# B&R Automation Studio project Soiled_PLC (part 11)

#### actGetServerReq.st
```iecst
(********************************************************************
 * COPYRIGHT --
 ********************************************************************
 * Program: hlKanLink
 * File: actGetServerReq.st
 * Author: stahlhut
 * Created: April 01, 2015
 ********************************************************************
 * Implementation of program hlKanLink
 ********************************************************************)

(* Kanlink Server/Request bearbeiten *)
ACTION actGetServerReq:
			// Commandos unter 1000 sind für alle gleich:
			IF Kanlink.ServerData.HeaderV1Rec.Command < 1000 THEN

				CASE Kanlink.ServerData.HeaderV1Rec.Command OF
					0:   // MaschinenInfo Senden: Darf jeder lesen

						Kanlink.ServerData.HeaderV1Send.Command := 1;
						Kanlink.ServerData.HeaderV1Send.dataFormat := 5;
						Kanlink.ServerData.HeaderV1Send.Length := 148;
						Kanlink.ServerData.HeaderV1Send.Tag := Kanlink.ServerData.HeaderV1Rec.Tag;
						Kanlink.ServerData.HeaderV1Send.ReqID := Kanlink.ServerData.HeaderV1Rec.ReqID;

						KLLib_SendData(ADR(Kanlink),ADR(Kanlink.ServerData.MetaInfoResp),SIZEOF(Kanlink.ServerData.MetaInfoResp),ADR(Kanlink.client_address));

					2:   // Response Ping: Darf jeder lesen

						Kanlink.ServerData.HeaderV1Send.Command := 3;
						Kanlink.ServerData.HeaderV1Send.dataFormat := 5;
						Kanlink.ServerData.HeaderV1Send.Length := 17;
						Kanlink.ServerData.HeaderV1Send.Tag := Kanlink.ServerData.HeaderV1Rec.Tag;
						Kanlink.ServerData.HeaderV1Send.ReqID := Kanlink.ServerData.HeaderV1Rec.ReqID;

						KLLib_SendData(ADR(Kanlink),ADR(Kanlink.ServerData.PingResp),SIZEOF(Kanlink.ServerData.PingResp),ADR(Kanlink.client_address));

				END_CASE;

			ELSE
					// >= 1000 sind spezifische Daten

					// Anfrage Konfiguriert?
					// Zur Anfrage Verbindung raussuchen..
					_xIdxFound := FALSE;
					_iIdxFound := 32000;

					KL_BuildKey(Command := Kanlink.ServerData.HeaderV1Rec.Command,CmdNr := UINT_TO_USINT( Kanlink.ServerData.HeaderV1Rec.CmdNr AND 16#000F) ,IPAdr := Kanlink.ServerData.IPAdr, adrKey:= ADR(Kanlink.RecKey));
					FOR _i := 0 TO HLKANLINK_MAX_SERVERCONNS  DO

						_ptrIndex ACCESS ADR(Kanlink.ServerListe[_i]);
						_dSrvIf ACCESS _ptrIndex.adrInterface;
						IF _ptrIndex.Adr = 0 THEN // wenn alle das Commando lesen dürfen/ Adresse und Area ausblenden
							IF Kanlink.RecKey.CmdKey = _ptrIndex.Key.CmdKey THEN // Index gefunden, beantworten:
								_xIdxFound := TRUE;
								_iIdxFound := _i;
								EXIT;
							END_IF;
						ELSE
							IF (Kanlink.RecKey.CmdKey = _ptrIndex.Key.CmdKey) AND (Kanlink.RecKey.IP_Key = _ptrIndex.Key.IP_Key) THEN // Index gefunden, beantworten:
								_xIdxFound := TRUE;
								_iIdxFound := _i;
								EXIT;
							END_IF;
						END_IF;
					END_FOR

					_xAdrErr := (_ptrIndex.AdrDataReq = 0) OR (_ptrIndex.AdrDataResp = 0);

					IF ( _xIdxFound = FALSE) OR _xAdrErr THEN // Falls keine gültige Verbindung dann Fehlerframe senden
						// Fehlerframe senden:
						Kanlink.ServerData.HeaderV1Send.Command := Kanlink.ServerData.HeaderV1Rec.Command +1;
						Kanlink.ServerData.HeaderV1Send.dataFormat := 255;
						Kanlink.ServerData.HeaderV1Send.Length := 68;
						Kanlink.ServerData.HeaderV1Send.Tag := Kanlink.ServerData.HeaderV1Rec.Tag;
						Kanlink.ServerData.HeaderV1Send.ReqID := Kanlink.ServerData.HeaderV1Rec.ReqID;

						// Error Frame:
						Kanlink.ServerData.ErrorFrame.ErrorNumber := 2;
						strcpy(ADR(Kanlink.ServerData.ErrorFrame.ErrorText),ADR('request not supported'));

						//	KLLib_SendData(ADR(Kanlink),ADR(Kanlink.ServerData.ErrorFrame),SIZEOF(Kanlink.ServerData.ErrorFrame),ADR(Kanlink.client_address));

					ELSE
						// Empfangene Daten speichern:

						IF NOT( (_dSrvIf.iState <> 0 )   AND _ptrIndex.xReqManually) THEN  // falls Req bereits bearbeitet wird verwerfen
							_ptrIndex.iReqCnt := _ptrIndex.iReqCnt + 1;
							_dSrvIf.iState := 1;
							strcpy(ADR(_ptrIndex.sClientIPAdr),ADR(Kanlink.client_address));
							// todo längenüberprüfung _ptrIndex.ReqLength
							memcpy(_ptrIndex.AdrDataReq,ADR(Kanlink.ServerData.receive_data)+PreHeaderSize+HeaderSize,_ptrIndex.ReqLength);

							_ptrIndex.iReqID := Kanlink.ServerData.HeaderV1Rec.ReqID;
							_dSrvIf.out.tag		:= Kanlink.ServerData.HeaderV1Rec.Tag;

							IF (_ptrIndex.CmdOpt AND KL_optOnReqCall) <> 0 THEN
								KL_OnRecReq(adrReqData := _ptrIndex.AdrDataReq, adrRespData := _ptrIndex.AdrDataResp, adrKanlink := ADR(Kanlink),_ptrIndex.Cmd, adrUserData := IFhlKanLink.Parameter.adrUserTyp );
							END_IF;
							IF _ptrIndex.xReqManually = 0 THEN

								Kanlink.ServerData.HeaderV1Send.Command := _ptrIndex.Cmd + 1;
								Kanlink.ServerData.HeaderV1Send.dataFormat := 5;
								Kanlink.ServerData.HeaderV1Send.Length := UDINT_TO_UINT( _ptrIndex.RespLength);
								Kanlink.ServerData.HeaderV1Send.ReqID := _ptrIndex.iReqID;
								Kanlink.ServerData.HeaderV1Send.CmdNr := _ptrIndex.CmdOpt AND 16#000F;
								Kanlink.ServerData.HeaderV1Send.Tag		:= _dSrvIf.tag;
								_ptrIndex.iConnectionTimer := 0;
								KLLib_SendData(ADR(Kanlink),_ptrIndex.AdrDataResp,_ptrIndex.RespLength,ADR(_ptrIndex.sClientIPAdr));
							END_IF;
						END_IF;

					END_IF;

			END_IF;

END_ACTION
```

#### actResponse.st
```iecst
(********************************************************************
 * COPYRIGHT --
 ********************************************************************
 * Program: hlKanLink
 * File: actResponse.st
 * Author: stahlhut
 * Created: April 01, 2015
 ********************************************************************
 * Implementation of program hlKanLink
 ********************************************************************)

(* Response eines Servers bearbeiten *)
ACTION actResponse:

			KL_BuildKey(Command := Kanlink.ServerData.HeaderV1Rec.Command,CmdNr := UINT_TO_USINT( Kanlink.ServerData.HeaderV1Rec.CmdNr AND 16#000F) ,IPAdr := Kanlink.ServerData.IPAdr, adrKey:= ADR(Kanlink.RecKey));

			_xIdxFound := FALSE;
			FOR _i := 0 TO HLKANLINK_MAX_CLIENTCONNS DO
				_dClient ACCESS ADR(Kanlink.ClientListe[_i]);

				IF (Kanlink.RecKey.CmdKey = _dClient.Key.CmdKey) AND (Kanlink.RecKey.IP_Key = _dClient.Key.IP_Key) THEN // Index gefunden, beantworten:
					_xIdxFound := TRUE;
					EXIT;
				END_IF;
			END_FOR

			_xAdrOK := _dClient.AdrDataResp <> 0 ;

			IF _xIdxFound AND _xAdrOK THEN
				_dClient.xReqPending := FALSE;
				IF _dClient.iTimeOutCnt > 0 THEN
					_dClient.iTimeOutCnt := _dClient.iTimeOutCnt - 1;
				END_IF;
				IF _dClient.adrInterface <> 0 THEN
					_dCltIf ACCESS _dClient.adrInterface;
					_dCltIf.iState := 3;
				END_IF;

				memcpy(_dClient.AdrDataResp,ADR(Kanlink.ServerData.receive_data) + PreHeaderSize+HeaderSize,_dClient.RespLength);
				_dCltIf.out.recTag := Kanlink.ServerData.HeaderV1Rec.Tag;

		  	END_IF;

			_iCltRespCnt := _iCltRespCnt + 1;
			Kanlink._xGetClientResp := FALSE;

			Kanlink._xSendClient := TRUE; // Daten einsortiert, nix weiter zutun also Clients bearbeiten
			Kanlink.udp.rec.enable := 1;

END_ACTION
```

### history.txt
```
1.00.3 horn 20.03.2017
hlKanLink wurde so erweitert, dass jetzt beim Server und Client eine beliebige IP-Adresse eingegeben werden kann.
AdvMode		Freischalten der Eingabe der gesamten IP-Adresse
AdrAdvMode	gesamte IP-Adresse der Gegenstelle.

1.00.2 horn 20.01.2016
Es werden jetzt keine Warnmeldungen mehr erzeugt.

1.00.1 sta 1.4.2015 sta
KG Framework - Kompatibel
Der Client kann nun einen UDINT Tag zum Server senden. Unterstützt der Server den Tag
wird ein Server-Tag zurückgesendet.
ifhlKanlink

0.94.5 sta 16.12.2014
udp_open mit IP-Adresse binden
27.3.12/sta/Struktur für Visualisierung

20.3.12/sta/Kommando Typen in einzelne Dateien geteilt
Compiler schalter "Autonom" eingefügt, Lib Autonom erstellt
Cmd WetExt angepasst

7.3.12/sta/version Kgframework
hlKanlink Version

21.02.12 sta 0.93
Client kann mit state gesteuert werden

8.2.12 sta 0.92
Fehler bei Server-Key behoben
2.2.12 sta
Zum einrichten eines Server und Client KLLib_CfgServer und KLLib_CfgClient integriert.
Konf sowohl über Parameter und mit den Funktionen möglich

30.1.12 sta
interface  umbenannt
MaxServerConn und MaxClientCon in userlib

todo:
"OneShot" Client-Statevariable
Überprüfung Längen der Commandos
Logger wieder inbetriebnehmen

Startversion 0.900
```

### Library Logical/KanLink_A19/KGFramework/Pkg_hlKanLink/KanLinkLib (IEC, version 0.94.5) - KanlinkHilfsfunktionen
Depends on: AsUDP, asstring, AsARCfg, brsystem, sys_lib, AsArLog, AsIODiag, AsETH, DataObj, KL_UserLib, KGstdLib

#### CmdBTxfer.typ - Commando Batch Transfer
```iecst
(********************************************************************
 * COPYRIGHT -- Herbert Kannegiesser GmbH
 ********************************************************************
 * Library: Kanlink Commando 1000 BatchTransfer
 * File:
 * Author: stahlhut
 * Created: 20.03.2012
 ********************************************************************
 * Data types of library WetLinkLib
 ********************************************************************)
(*Interne Strukturen*)

TYPE
	KL_BTxf_typ : 	STRUCT  (*Batch Transfer Server*)
		Req : KLreq1000_BTH_typ;
		Resp : KLresp1000_BTH_typ;
	END_STRUCT;
	KLreq1000_BTH_typ : 	STRUCT
		xHready : BOOL;
		xHreadyForLoad : BOOL;
		xHbatchReceived : BOOL;
		xHtransferzoneOccupied : BOOL;
		xHreqCtrlTransfer : BOOL;
		xHtransferRunning : BOOL;
		xHwaitingForTransfer : BOOL;
		xHshiftBatches : BOOL;
		wHstate : UINT;
		xHcmdAutomatic : BOOL;
		xHreserve : ARRAY[1..5]OF BOOL;
		wTimeToReadyForLoad : UINT;
		wRemainProctime : UINT; (*Remaining Processtime / Verbleibende Prozesszeit*)
	END_STRUCT;
	KLresp1000_BTH_typ : 	STRUCT
		xHsCmdFinishProcess : BOOL;
		xHsReqForUnload : BOOL;
		xHsUnloading : BOOL;
		xHsReqCtrlTransfer : BOOL;
		xHsTransferRunning : BOOL;
		xHsRes : BOOL;
		wState : UINT;
		xCmdAuto : BOOL;
		xCmdStartProcess : BOOL;
		xHsDataValid : BOOL;
		xHsRes2 : ARRAY[0..2]OF BOOL;
		wCntLoads : UINT;
		BatchData : BatchData_typ;
	END_STRUCT;
END_TYPE
```

#### KLInterface.typ - Interfacetypen Kanlink
```iecst
(********************************************************************
 * COPYRIGHT -- Herbert Kannegiesser GmbH
 ********************************************************************
 * Library: Kanlink	 Interface
 * File:
 * Author: stahlhut
 * Created: 20.03.2012
 ********************************************************************
 * Data types of Interface Kanlink
 ********************************************************************)

TYPE
	KL_Key_typ : 	STRUCT
		IP_Key : UDINT;
		CmdKey : UDINT;
	END_STRUCT;
	KL_Parameter_typ : 	STRUCT
		Server : ARRAY[0..HLKANLINK_MAX_SERVERCONNS]OF KL_ServerPar_typ;
		Client : ARRAY[0..HLKANLINK_MAX_CLIENTCONNS]OF KL_ClientPar_typ;
		adrUserTyp : UDINT;
	END_STRUCT;
	KL_ClientPar_typ : 	STRUCT
		Name : STRING[15];
		Adr : UINT;
		Cmd : UINT;
		CmdOpt : UINT; (*Bits 0..3 = Nummer des Clients*)
		Area : UINT;
		CycleTime : UINT;
		sReq : STRING[80];
		sResp : STRING[80];
		AdvMode : BOOL; (*Modus mit dem eine vollständige IP-Adresse eingegeben werden kann*)
		AdrAdvMode : STRING[16]; (*Vollständige IP-Adresse*)
	END_STRUCT;
	KL_ServerPar_typ : 	STRUCT
		Name : STRING[15];
		Adr : UINT;
		Cmd : UINT;
		CmdOpt : UINT; (*Bits 0..3 = Nummer der Verbindung*)
		Area : UINT;
		TimeOut : UINT;
		sReq : STRING[80];
		sResp : STRING[80];
		AdvMode : BOOL; (*Modus mit dem eine vollständige IP-Adresse eingegeben werden kann
oder die Prüfung der IP-Adresse entfällt.*)
		AdrAdvMode : STRING[16]; (*Vollständige IP-Adresse*)
	END_STRUCT;
	IF_ServerOutTyp : 	STRUCT
		xConnected : BOOL;
		iCfgState : UINT; (*0 = ConfOK*)
		tag : UDINT;
	END_STRUCT;
	IF_Server_typ : 	STRUCT
		iState : UINT;
		out : IF_ServerOutTyp;
		tag : UDINT;
	END_STRUCT;
	IF_ClientOut_typ : 	STRUCT
		xConnected : BOOL;
		recTag : UDINT;
	END_STRUCT;
	IF_Client_typ : 	STRUCT
		out : IF_ClientOut_typ;
		iState : UINT;
		tag : UDINT;
	END_STRUCT;
	IFhlKanLink_Typ : 	STRUCT
		in : IF_KL_Control_in_typ;
		Server : ARRAY[0..HLKANLINK_MAX_SERVERCONNS]OF IF_Server_typ;
		Client : ARRAY[0..HLKANLINK_MAX_CLIENTCONNS]OF IF_Client_typ;
		Parameter : KL_Parameter_typ;
		xError : BOOL; (*Kanlink in Störung*)
	END_STRUCT;
	IF_KL_Control_in_typ : 	STRUCT
		xRun : BOOL; (*Rise= Starten Kanlink /fall = stoppen Kanlink*)
		xRestart : BOOL;
	END_STRUCT;
	IF_KL_Control_out_typ : 	STRUCT
		iError : UINT;
		iServerError : ARRAY[0..HLKANLINK_MAX_SERVERCONNS]OF UINT;
		iClientError : ARRAY[0..HLKANLINK_MAX_CLIENTCONNS]OF UINT;
		iStep : UINT; (*Statemachine KanLink*)
	END_STRUCT;
	IFhlKLVisuIN_typ : 	STRUCT
		cmdNr : INT; (*Ausführbares Commando*)
		cmdTag : INT; (*Dazugehörige Daten*)
		iServerNr : UINT; (*zu lesende Serverlist*)
		iCltNr : UINT; (*zu lesender Client*)
	END_STRUCT;
	IFhlKLVisuOUT_typ : 	STRUCT
		step : UINT;
		udpOpenStatus : UINT;
		udpSendStatus : UINT;
		udpRecStatus : UINT;
		iCycleTime : UINT;
		udNetId : UDINT;
		server : KL_ServerListe_typ;
		client : KL_ClientListe_typ;
		cmdResp : INT; (*Response auf CmdNr*)
	END_STRUCT;
	IFhlKLVisu_typ : 	STRUCT
		in : IFhlKLVisuIN_typ;
		out : IFhlKLVisuOUT_typ;
	END_STRUCT;
END_TYPE
```

#### KanLinkLib.typ - Exported data types
```iecst
(********************************************************************
 * COPYRIGHT -- Herbert Kannegiesser GmbH
 ********************************************************************
 * Library: WetLinkLib
 * File: WetLinkLib.typ
 * Author: stahlhut
 * Created: January 06, 2012
 ********************************************************************
 * Data types of library WetLinkLib
 ********************************************************************)
(*Interne Strukturen*)

TYPE
	udp_typ : 	STRUCT  (*UDP Typ*)
		open : UdpOpen;
		send : UdpSend;
		rec : UdpRecv;
		close : UdpClose;
	END_STRUCT;
	udint_array_typ : 	STRUCT  (*Casten von UDINT -> byte*)
		a : USINT;
		b : USINT;
		c : USINT;
		d : USINT;
	END_STRUCT;
	ServerDataTyp : 	STRUCT  (*Datatyp for global Variables*)
		receive_data : ARRAY[0..8191]OF USINT; (*Data which has been received*)
		send_data : ARRAY[0..8191]OF USINT; (*Data which should be sent*)
		PreHeaderSend : PreHeader_Typ;
		PreHeaderRec : PreHeader_Typ;
		HeaderV1Send : HeaderV1_Typ;
		HeaderV1Rec : HeaderV1_Typ;
		MetaInfoResp : KLresp0_MetaInfo_typ;
		ErrorFrame : KL_Error_Frame_typ;
		PingReq : KLreq2_Ping_typ;
		PingResp : KLresp2_Ping_typ;
		IPAdr : STRING[16]; (*IP-Adresse des Clients*)
	END_STRUCT;
	PreHeader_Typ : 	STRUCT
		Magic : UDINT; (*MagicNr*)
		HeaderVersion : UINT; (*Headerversion*)
		Tag : UINT; (*Reserve*)
	END_STRUCT;
	HeaderV1_Typ : 	STRUCT
		ReqID : UINT;
		dataFormat : UINT;
		Command : UINT;
		Length : UINT;
		CmdNr : UINT;
		CmdTag : UINT; (*Unterschiedliche Parameter zum Command*)
		Tag : UDINT; (*Reserve/Spezial*)
	END_STRUCT;
	KL_ServerListe_typ : 	STRUCT
		Cmd : UINT;
		CmdOpt : UINT;
		Adr : UINT;
		Area : UINT;
		pRespStr : UDINT; (*Adresse des Resp String*)
		pReqStr : UDINT; (*Adresse des Req String*)
		AdrDataReq : UDINT;
		ReqLength : UDINT; (*Länge Request Daten*)
		AdrDataResp : UDINT;
		RespLength : UDINT; (*Länge Response Daten*)
		Key : KL_Key_typ; (*Suchschlüssel/ Darf nicht doppelt vorkommen== Konfigurierungsfehler*)
		xConnected : BOOL; (*Falls Commando 2s nicht angefragt wird ist verbindung unterbrochen*)
		iConnectionTimer : UINT; (*Der Zugehörige Zähler / Timer*)
		adrParameter : UDINT; (*Adresse der Parameter*)
		sServerIPAdr : STRING[16];
		sClientIPAdr : STRING[16];
		iReqCnt : UINT;
		xReqManually : BOOL;
		iReqID : UINT;
		iCfgStatus : UINT;
		adrInterface : UDINT;
		xActiv : BOOL;
		tag : UDINT;
	END_STRUCT;
	KL_ClientListe_typ : 	STRUCT
		RecCmd : UINT; (*Rec Command nr*)
		Cmd : UINT; (*Send Command nr*)
		CmdOpt : UINT; (*SendeOptionen Senden Nr des Commando etc*)
		Adr : UINT;
		Area : UINT;
		Key : KL_Key_typ;
		pResp : UDINT; (*Adresse des Namen der Response Struktur*)
		pReq : UDINT; (*Adresse des Namen der Request Struktur*)
		AdrDataReq : UDINT;
		AdrDataResp : UDINT;
		ReqLength : UDINT;
		RespLength : UDINT;
		TimeOut : UINT;
		TimeOutLeft : UINT;
		xError : BOOL;
		iCycleWait : UINT;
		iCycleTime : UINT;
		xDataRec : BOOL;
		iReqId : UINT;
		sClientAdr : STRING[16];
		xReqPending : BOOL;
		iTimeOutCnt : UINT;
		xActiv : BOOL;
		iCnt : UINT;
		xConnected : BOOL; (*True wenn Verbindung aktiv und läuft*)
		iTimeOutCnt_Summe : UINT;
		adrInterface : UDINT;
		adrParameter : UDINT; (*Adresse der Parameter*)
		recTag : UDINT; (*Tag des Kommandos*)
	END_STRUCT;
END_TYPE

(*Kommandos*)

TYPE
	BatchData_typ : 	STRUCT
		dtTimeStamp : DATE_AND_TIME;
		bTypeBatchNo : USINT;
		bCntCustomers : USINT;
		wTotalWeight : UINT;
		bBatchNo : ARRAY[0..15]OF USINT;
		sCategory : STRING[11];
		utfMark : ARRAY[0..31]OF UINT;
		bCustom : ARRAY[0..11]OF USINT;
		PartBatch : ARRAY[0..7]OF PartBatchData_typ;
	END_STRUCT;
	PartBatchData_typ : 	STRUCT
		sCustomNo : STRING[11];
		wCustomWeight : UINT;
	END_STRUCT;
	KL_Error_Frame_typ : 	STRUCT
		Version : UINT;
		ErrorNumber : UINT;
		ErrorText : STRING[63];
	END_STRUCT;
	KLresp0_MetaInfo_typ : 	STRUCT
		KanLink_Hostname : STRING[15];
		Machine_type : STRING[15];
		SoftwareNo : STRING[15];
		SoftwareVersion : STRING[15];
		DataModelTimeStamp : DATE_AND_TIME;
		DataModelVersion : UINT;
		TimeZone : UINT;
		SommerTime : UINT;
	END_STRUCT;
	KLreq2_Ping_typ : 	STRUCT
		KanLink_Hostname : STRING[15];
	END_STRUCT;
	KLresp2_Ping_typ : 	STRUCT
		KanLink_Hostname : STRING[15];
		FrameVersion : USINT;
	END_STRUCT;
END_TYPE
```

#### KanLinkLib.fun - Exported functions and function blocks
```iecst
(********************************************************************
 * COPYRIGHT -- Herbert Kannegiesser GmbH
 ********************************************************************
 * Library: WetLinkLib
 * File: WetLinkLib.fun
 * Author: stahlhut
 * Created: January 06, 2012
 ********************************************************************
 * Functions and function blocks of library WetLinkLib
 ********************************************************************)

FUNCTION_BLOCK KanLink_FB (*TODO: Add your comment here*)
	VAR_INPUT
		Step : UINT; (*state machine*)
		ErrorNr : UINT;
		client_address : STRING[16]; (*Speichern der Receiver Adresse*)
		RecKey : KL_Key_typ;
		sNetID : STRING[15];
		udNetID : UDINT;
		udp : udp_typ;
		ServerData : ServerDataTyp;
		ServerListe : ARRAY[0..HLKANLINK_MAX_SERVERCONNS] OF KL_ServerListe_typ; (*Erlaubte Daten Server*)
		ClientListe : ARRAY[0..HLKANLINK_MAX_CLIENTCONNS] OF KL_ClientListe_typ;
		_xOpenPort : BOOL;
		_xSendClient : BOOL;
		_xGetClientResp : BOOL;
		_xGetServerReq : BOOL;
		_uiLastId : UDINT;
		CanReturn : BOOL;
		adrSelf : UDINT; (*Eigene Adresse, zum weiterleiten an Function/Function Block*)
		_offset : UDINT; (*Offset zum Berechnen der Sendelänge*)
		_SendLen : UDINT; (*Sendelänge*)
		DoCommand : UINT;
		KLLib_Init_0 : KLLib_Init;
		_iCycleTime : UINT;
		adrInterface : UDINT;
		iPort : UINT; (*Port nr (23500)*)
		sIF : STRING[10]; (*Interface Ethernet*)
		CfgClient : KLLib_CfgClient;
		CfgServer : KLLib_CfgServer;
	END_VAR
	VAR_OUTPUT
		xReturn : BOOL;
	END_VAR
	VAR
		_dPrehead : REFERENCE TO PreHeader_Typ;
		_dHead : REFERENCE TO HeaderV1_Typ;
		_udArr : REFERENCE TO udint_array_typ;
		_dRecAdr : UDINT;
		_xPreheadOK : BOOL;
		_xVersionOK : BOOL;
		_xUse : BOOL;
	END_VAR
END_FUNCTION_BLOCK

FUNCTION KLLib_ClientTimer : BOOL (*Bearbeitet Timeout und Cycletime (Zähler)*)
	VAR_INPUT
		Srv : REFERENCE TO KanLink_FB;
		_iCycleTime : UINT;
	END_VAR
	VAR
		_dClient : REFERENCE TO KL_ClientListe_typ;
		_i : UINT;
		_dServer : REFERENCE TO KL_ServerListe_typ;
		_dInterface : REFERENCE TO IF_Client_typ;
		_dSrvIf : REFERENCE TO IF_Server_typ;
	END_VAR
END_FUNCTION

FUNCTION KLLib_GetPVAdr : UDINT (*Adresse der PV ermitteln (Server)*)
	VAR_INPUT
		ServerItem : REFERENCE TO KL_ServerListe_typ;
	END_VAR
	VAR
		iStat : INT;
	END_VAR
END_FUNCTION

FUNCTION KLLib_SendData : UDINT (*TODO: Add your comment here*)
	VAR_INPUT
		Srv : REFERENCE TO KanLink_FB;
		SendAdr : UDINT;
		SendLen : UDINT;
		pDestination : UDINT; (*Adresse des Zielstrings*)
	END_VAR
END_FUNCTION

FUNCTION KLLib_ReadServerPara : UDINT (*TODO: Add your comment here*)
	VAR_INPUT
		adrServerItem : UDINT;
		adrParaItem : UDINT;
		adrKanLink : UDINT;
	END_VAR
	VAR
		_xError : BOOL;
		KanLink : REFERENCE TO KanLink_FB;
		dServer : REFERENCE TO KL_ServerListe_typ;
		dPara : REFERENCE TO KL_ServerPar_typ;
		_udAdr : UDINT;
		_udArr : REFERENCE TO udint_array_typ;
		_udNetId : REFERENCE TO udint_array_typ;
	END_VAR
END_FUNCTION

FUNCTION KLLib_ReadClientPara : UDINT (*TODO: Add your comment here*)
	VAR_INPUT
		adrClientItem : UDINT;
		adrParaItem : UDINT;
		adrServer : UDINT;
	END_VAR
	VAR
		_xError : BOOL;
		dClient : REFERENCE TO KL_ClientListe_typ;
		dPara : REFERENCE TO KL_ClientPar_typ;
		_udArr : REFERENCE TO udint_array_typ;
		_udAdr : UDINT;
		dServer : REFERENCE TO KanLink_FB;
		_udNetId : REFERENCE TO udint_array_typ;
	END_VAR
END_FUNCTION

FUNCTION KLLib_InitCltPV : UDINT (*TODO: Add your comment here*)
	VAR_INPUT
		dclt : REFERENCE TO KL_ClientListe_typ;
	END_VAR
	VAR
		iStat : UINT;
	END_VAR
END_FUNCTION

FUNCTION_BLOCK KLLib_Init (*TODO: Add your comment here*)
	VAR_INPUT
		enable : BOOL;
		adrServer : UDINT;
		adrInterface : UDINT;
	END_VAR
	VAR_OUTPUT
		status : UINT;
	END_VAR
	VAR
		_bStep : INT;
		_dServer : REFERENCE TO KanLink_FB;
		GetEthPort_0 : kgGetEthPort;
		CfgGetIPAddr_0 : CfgGetIPAddr;
		RTInfo_0 : RTInfo;
		_i : INT;
		_dIf : REFERENCE TO IFhlKanLink_Typ;
	END_VAR
END_FUNCTION_BLOCK

FUNCTION KL_BuildKey : BOOL
	VAR_INPUT
		Command : UINT;
		CmdNr : USINT;
		IPAdr : STRING[16];
		adrKey : UDINT;
	END_VAR
	VAR
		IP_Key : UDINT;
		Key : REFERENCE TO KL_Key_typ;
	END_VAR
END_FUNCTION

FUNCTION_BLOCK KLLib_CfgClient (*Configuriert einen Kanlink Client*)
	VAR_INPUT
		adrKanlink : UDINT;
		ClientIndex : UINT;
		adrName : UDINT;
		IPAdr : USINT;
		Area : USINT;
		CmdOpt : UINT;
		Cmd : UINT;
		CycleTime : UINT;
		adrSReq : UDINT;
		adrSResp : UDINT;
	END_VAR
	VAR_OUTPUT
		status : UINT;
	END_VAR
	VAR
		_dKL : REFERENCE TO KanLink_FB;
		_dCltPar : REFERENCE TO KL_ClientPar_typ;
		_iret : UDINT;
	END_VAR
END_FUNCTION_BLOCK

FUNCTION_BLOCK KLLib_CfgServer (*Configuriert einen Kanlink Server*)
	VAR_INPUT
		adrKanlink : UDINT;
		ServerIndex : UINT;
		adrName : UDINT;
		IPAdr : USINT;
		Area : USINT;
		CmdOpt : UINT;
		Cmd : UINT;
		TimeOut : UINT;
		adrSReq : UDINT;
		adrSResp : UDINT;
	END_VAR
	VAR_OUTPUT
		status : UINT;
	END_VAR
	VAR
		_dKL : REFERENCE TO KanLink_FB;
		_dSrvPar : REFERENCE TO KL_ServerPar_typ;
		_iret : UDINT;
	END_VAR
END_FUNCTION_BLOCK

FUNCTION KLLib_CreateStrucDef : UINT (*Erzeuge eine Strukturdefinition zu einer Variablen*)
	VAR_INPUT
		lPtrAdr : UDINT;
		lPtrLen : UDINT;
		sRootName : STRING[127];
		sItemName : STRING[31];
		lDataAdr : UDINT;
	END_VAR
	VAR
		_wStatus : UINT;
		_sPvName : STRING[127];
		_lDataType : UDINT;
		_lDataLen : UDINT;
		_wDataDimension : UINT;
		_sLine : STRING[127];
		_sValueLen : STRING[11];
		_lAdr : REFERENCE TO UDINT;
		_lLen : REFERENCE TO UDINT;
		_sValueDim : STRING[5];
		_sValueOffs : STRING[11];
		_i : UINT;
		_sItemName : STRING[31];
		_sType : ARRAY[1..23] OF STRING[15] := ['BOOL','SINT','INT','DINT','USINT','UINT','UDINT','REAL','STRING','ULINT','DATE_AND_TIME','TIME','DATE','LREAL','','TIME_OF_DAY','BYTE','WORD','DWORD','LWORD','WSTRING','','LINT'];
		_lDataAdr : UDINT;
	END_VAR
END_FUNCTION

FUNCTION KLLib_WriteStrucDefLine : UINT (*Übertrage einen String als Zeile in den Speicher*)
	VAR_INPUT
		lPtrLine : UDINT;
		lPtrAdr : UDINT;
		lPtrLen : UDINT;
	END_VAR
	VAR
		_lAdr : REFERENCE TO UDINT;
		_lLen : REFERENCE TO UDINT;
		_iStringlen : INT;
		_sLine : REFERENCE TO STRING[127];
	END_VAR
END_FUNCTION
```

#### KanLink_FB.st - core-Funktion
```iecst
(********************************************************************
 * COPYRIGHT -- Herbert Kannegiesser GmbH
 ********************************************************************
 * Library: Kanlink
 * File:
 * Author: stahlhut
 * Created: January 06, 2012
 ********************************************************************
 * Implementation of library Kanlink

29.8.2012 Bug behoben verunden recAdr mit 0x0F

 ********************************************************************)

FUNCTION_BLOCK KanLink_FB

	xReturn := 0;

	IF Step <> 10 THEN
		xReturn := 1;
		RETURN;
	END_IF;
	KLLib_ClientTimer(adrSelf,_iCycleTime);

	IF  udp.send.enable THEN
		udp.send;

		IF  udp.send.status = 0 THEN
			udp.send.enable := FALSE;
		ELSIF udp.send.status = ERR_FUB_BUSY THEN
			udp.send.enable := TRUE;
			xReturn := 1;
			RETURN;
		ELSE
			ErrorNr := 4;
			udp.send.enable := FALSE;
		END_IF
	END_IF;

	udp.rec.enable := 1;
	udp.rec.ident := udp.open.ident;
	udp.rec.pData := ADR(ServerData.receive_data);	// Datenspeicher
	udp.rec.datamax := SIZEOF(ServerData.receive_data);	// Länge des Datenspeichers
	udp.rec.flags := 0;
	udp.rec.pIpAddr := ADR(client_address);	// IP Adresse des Senders
	udp.rec;

	IF udp.rec.status = 0 THEN  // Daten empfangen
		// Header Daten kopieren
		_dPrehead ACCESS ADR(ServerData.receive_data);
		_dHead ACCESS ADR(ServerData.receive_data) + PreHeaderSize;
		memcpy(ADR(ServerData.PreHeaderRec),ADR(ServerData.receive_data),PreHeaderSize);
		memcpy(ADR(ServerData.HeaderV1Rec),ADR(ServerData.receive_data)+PreHeaderSize,SIZEOF(ServerData.HeaderV1Rec));

		ServerData.IPAdr := client_address;

		_xPreheadOK := (ServerData.PreHeaderRec.Magic = MagicNr);
		_xVersionOK := (ServerData.PreHeaderRec.HeaderVersion = 16#100);

		IF (_dHead.Command AND 1) = 0 THEN
			_xGetServerReq := TRUE;
		ELSIF (_dHead.Command AND 1) = 1 THEN
			_xGetClientResp := TRUE;
		END_IF;

	ELSIF udp.rec.status = udpERR_NO_DATA THEN  // Keine Daten empfangen, Client abarbeiten
		_xSendClient := TRUE;
	ELSIF udp.rec.status = ERR_FUB_BUSY THEN  (* UdpRecv not finished -> redo *)
		xReturn := 1;
		RETURN;
	ELSE  (* Goto Error Step *)
		ErrorNr := 5;
		xReturn := 1;
		RETURN;
	END_IF

	// dieser teil ist nur für den Linker (unused Variable)
	IF _xUse THEN
		RecKey := RecKey;
		sNetID := sNetID;
		udNetID := udNetID;
		ServerListe := ServerListe;
		ClientListe	:= ClientListe;
		_xOpenPort := _xOpenPort;
		_uiLastId	:= _uiLastId;
		CanReturn	:= CanReturn;
		_offset 	:= _offset;
		_SendLen	:= _SendLen;
		DoCommand	:= DoCommand;
	 	adrInterface	:= adrInterface;
		iPort 	:= iPort;
		sIF	:= sIF;
		KLLib_Init_0.enable	:= KLLib_Init_0.enable;
		CfgClient.adrKanlink	:= CfgClient.adrKanlink;
		CfgServer.adrKanlink	:= CfgServer.adrKanlink;
	END_IF;

END_FUNCTION_BLOCK
```

#### KLLib_ClientTimer.st
```iecst
(********************************************************************
 * COPYRIGHT -- Herbert Kannegiesser GmbH
 ********************************************************************
 * Library: WetLinkLib
 * File: WLLIb_ClientTimer.st
 * Author: stahlhut
 * Created: January 06, 2012
 ********************************************************************
 * Implementation of library WetLinkLib
 ********************************************************************)

(* TODO: Add your comment here *)
FUNCTION KLLib_ClientTimer
FOR _i := 0 TO HLKANLINK_MAX_CLIENTCONNS DO
	_dClient  ACCESS ADR(Srv.ClientListe[_i]);
	_dInterface ACCESS (_dClient.adrInterface);

	// TimeOut (kurz) taskgerecht berechnen
	IF (_dClient.TimeOutLeft >= _iCycleTime) AND _dClient.xReqPending THEN
 		_dClient.TimeOutLeft := _dClient.TimeOutLeft - _iCycleTime;
	END_IF;

	IF _dClient.iCycleWait <= _dClient.iCycleTime THEN
		_dClient.iCycleWait := _dClient.iCycleWait + _iCycleTime;
	END_IF;
	// Timeout aufgetreten nur bis n Zählen. Retry sofort nach timeout, sonst retry nach cycletime
	IF _dClient.xReqPending AND (_dClient.TimeOutLeft < _iCycleTime) THEN
		_dClient.iTimeOutCnt_Summe := _dClient.iTimeOutCnt_Summe + 1;
		_dClient.xReqPending := FALSE;	// noch mal versuchen
		IF _dClient.iTimeOutCnt < 5 THEN
			_dClient.iTimeOutCnt := _dClient.iTimeOutCnt +1 ;
			_dClient.xReqPending := FALSE;	// noch mal versuchen
			_dInterface.iState := 4;
			_dClient.iCycleWait := _dClient.iCycleTime;
		END_IF;
	END_IF;
		// Verbindungsfehler
	_dClient.xConnected := (_dClient.iTimeOutCnt < 5) AND _dClient.xActiv AND (_dClient.iCycleTime > 0);
	_dInterface.out.xConnected := _dClient.xConnected;
	IF (_dClient.iTimeOutCnt >= 5 ) AND ( _dInterface.iState = 2 ) THEN
		_dInterface.iState := 255; // Timeout melden
	END_IF;

END_FOR;

FOR _i := 0 TO HLKANLINK_MAX_SERVERCONNS DO
	_dServer ACCESS ADR(Srv.ServerListe[_i]);
	_dSrvIf ACCESS _dServer.adrInterface;

	IF _dServer.iConnectionTimer <= 2000 THEN
		_dServer.iConnectionTimer := _dServer.iConnectionTimer + _iCycleTime;
	END_IF;
	_dServer.xConnected := (_dServer.iConnectionTimer < 2000);
	_dSrvIf.out.xConnected := _dServer.xConnected;
END_FOR;
KLLib_ClientTimer := 0;

END_FUNCTION
```

#### KLLib_SendData.st
```iecst
(********************************************************************
 * COPYRIGHT -- Herbert Kannegiesser GmbH
 ********************************************************************
 * Library: WetLinkLib
 * File: WLLib_SendData.st
 * Author: stahlhut
 * Created: January 07, 2012
 * changed April 2015
 ********************************************************************
 *
 ********************************************************************)

FUNCTION KLLib_SendData
	IF Srv.udp.send.enable = TRUE THEN //Sendung noch unterwegs, abbrechen
 		KLLib_SendData := 1;
		RETURN;
	END_IF;

	Srv.ServerData.PreHeaderSend.Magic := MagicNr;
	Srv.ServerData.PreHeaderSend.HeaderVersion := 16#0100;
	Srv._offset := 0;
	memcpy(ADR(Srv.ServerData.send_data),ADR(Srv.ServerData.PreHeaderSend),PreHeaderSize);
	Srv._offset := PreHeaderSize;

	memcpy(ADR(Srv.ServerData.send_data)+Srv._offset,ADR(Srv.ServerData.HeaderV1Send),HeaderSize);
	Srv._offset := Srv._offset+ HeaderSize;
	memcpy(ADR(Srv.ServerData.send_data)+Srv._offset,SendAdr,SendLen);
	Srv._SendLen := Srv._offset + Srv.ServerData.HeaderV1Send.Length;

	// Telegramm jetzt senden
	Srv.udp.send.enable := 1;
	Srv.udp.send.ident 	:= Srv.udp.open.ident;	(* Client Ident from AsUDP.UDP_Open *)
	Srv.udp.send.pHost 	:= pDestination;	(* IP Address of the Client *)
	Srv.udp.send.port 	:= Srv.iPort;
	Srv.udp.send.pData 	:= ADR(Srv.ServerData.send_data);	(* Which data to send *)
	Srv.udp.send.datalen :=  Srv._SendLen; //
	Srv.udp.send.flags 	:= 0;
	Srv.udp.send ;	(* Call the Function*)

END_FUNCTION
```

#### KL_BuildKey.st - Berechnen des Connection Key
```iecst
(********************************************************************
 * COPYRIGHT -- Herbert Kannegiesser GmbH
 ********************************************************************
 * Library: KanLinkLib
 * Datei: KL_BuildKey.st
 * Autor: stahlhut
 * Erstellt: 16. Januar 2012
 ********************************************************************
 * Implementierung der Library KanLinkLib
 ********************************************************************)

(* Berechnen des Connection Key *)
FUNCTION KL_BuildKey

	IF adrKey = 0 THEN // Fehler aufgetreten

		Key.CmdKey := 0;
		Key.IP_Key := 0;
		KL_BuildKey := FALSE;

	ELSE

		Key ACCESS adrKey;
		Key.CmdKey := SHL(UINT_TO_UDINT(Command),4)+USINT_TO_UINT(CmdNr);
		ethInetAton(ADR(IPAdr),ADR(IP_Key));
		Key.IP_Key := IP_Key;
		KL_BuildKey := TRUE;

	END_IF

END_FUNCTION
```

#### KLLib_Init.st
```iecst
(********************************************************************
 * COPYRIGHT -- Herbert Kannegiesser GmbH
 ********************************************************************
 * Library: KanLinkLib
 * File: KL_Init.st
 * Author: stahlhut
 * Created: January 12, 2012
 ********************************************************************
 * Implementation of library KanLinkLib
 ********************************************************************)

(* TODO: Add your comment here *)
FUNCTION_BLOCK KLLib_Init

	IF (adrServer = 0) OR (adrInterface = 0 )  THEN // fehler
		status := 1;
		enable := 0;
		RETURN;
	END_IF;
	IF enable = 0 THEN
		status := ERR_FUB_ENABLE_FALSE;
		RETURN;
	END_IF;

	IF (status = ERR_FUB_BUSY	) AND (enable = 0) THEN
		status := ERR_FUB_ENABLE_FALSE;
		_bStep := 100;
	END_IF;

	CASE _bStep OF
		0: // nix tun
			status := ERR_FUB_BUSY;
			_bStep := 10;
		10:
			_dServer ACCESS adrServer;
			_dServer.adrSelf := adrServer;
			_dIf ACCESS adrInterface;
			_dServer.adrInterface := adrInterface;

			IF _dServer.iPort = 0 THEN
				_dServer.iPort := 23500; // standardport benutzen
			END_IF;
			RTInfo_0.enable := TRUE;
			RTInfo_0;

			_dServer._iCycleTime := UDINT_TO_UINT( RTInfo_0.cycle_time / 1000);

			_bStep := 20;
		20:
			GetEthPort_0.enable := 1;
			GetEthPort_0.adrIF := ADR(_dServer.sIF);
			GetEthPort_0;
			IF GetEthPort_0.status = ERR_OK THEN
				_bStep := 30;
			ELSIF GetEthPort_0.status <> ERR_FUB_BUSY THEN // fehler aufgetreten
				status := 2;
				_bStep := 100;
			END_IF;
		30:
			CfgGetIPAddr_0.enable  := 1;
			CfgGetIPAddr_0.pDevice := ADR(_dServer.sIF);
			CfgGetIPAddr_0.pIPAddr := ADR(_dServer.sNetID);
			CfgGetIPAddr_0.Len := 16;
			CfgGetIPAddr_0;
			IF  (CfgGetIPAddr_0.status = ERR_OK) THEN
				_bStep := 40;
				ethInetAton(ADR(_dServer.sNetID),ADR(_dServer.udNetID));

			ELSIF CfgGetIPAddr_0.status <> ERR_FUB_BUSY THEN // fehler aufgetreten
				status := 3;
				_bStep := 100;
			END_IF;

		40:
			FOR _i := 0 TO HLKANLINK_MAX_SERVERCONNS DO
				_dServer.ServerListe[_i].adrInterface := ADR(_dIf.Server[_i]);
				KLLib_ReadServerPara(ADR(_dServer.ServerListe[_i]), ADR( _dIf.Parameter.Server[_i]),ADR(_dServer));
			END_FOR;
			//			memset(ADR(_dServer.ClientListe),0,SIZEOF(_dServer.ClientListe));
			FOR _i := 0 TO HLKANLINK_MAX_CLIENTCONNS DO
				KLLib_ReadClientPara(ADR(_dServer.ClientListe[_i]),ADR(_dIf.Parameter.Client[_i]),ADR(_dServer));
				_dServer.ClientListe[_i].xActiv := (_dServer.ClientListe[_i].Cmd <> 0);
				_dServer.ClientListe[_i].TimeOut := 140;
				_dServer.ClientListe[_i].adrInterface := ADR(_dIf.Client[_i]);
			END_FOR;
			_bStep := 50;
		50:

			_dServer.udp.open.enable := 1;
			_dServer.udp.open.pIfAddr := ADR(_dServer.sNetID);	(* Übergeben des Interface funzt nicht *)
			_dServer.udp.open.port := _dServer.iPort;	(* Port to listen*)
			_dServer.udp.open.options := 0;
			_dServer.udp.open;	(* Call the Function*)

			IF _dServer.udp.open.status = 0 THEN  (* UdpOpen successful*)
				_dServer._uiLastId := _dServer.udp.open.ident;
				_bStep := 90;
			ELSIF _dServer.udp.open.status = ERR_FUB_BUSY THEN  (* UdpOpen not finished -> redo *)

			ELSIF _dServer.udp.open.status = udpERR_ALREADY_EXIST THEN // erst schliessen
				_dServer.udp.close.enable := 1;
				_dServer.udp.close.ident := _dServer._uiLastId;
				_dServer.udp.close;
				IF _dServer.udp.close.status = 0 THEN
					//
				ELSIF _dServer.udp.close.status = ERR_FUB_BUSY THEN

				ELSE
					status := 5001;
					_bStep := 100;	// unbekannter close fehler aufgetreten
				END_IF;

			ELSE
				status := 5002;
				_bStep := 100; // unbekannter open fehler aufgetreten
			END_IF

		90:  // fertig
			status := ERR_OK;
			enable := 0;
			_bStep := 0;

		100: // fehler aufgetreten
			enable := 0;
			_bStep := 0;

	END_CASE;

END_FUNCTION_BLOCK
```

### Package Logical/KanLink_A19/KGFrameworkShare - Benutzereinstellungen


### Package Logical/KanLink_A19/KGFrameworkShare/Pkg_hlKanLinkUser - Kanlink User

### Library Logical/KanLink_A19/KGFrameworkShare/Pkg_hlKanLinkUser/KL_UserLib (IEC, version 0.91.0) - Kanlink User Library

#### KL_UserLib.var - Exported constants
```iecst
(********************************************************************
 * COPYRIGHT -- Herbert Kannegiesser GmbH
 ********************************************************************
 * Library: WL_UserLib
 * File: WL_UserLib.var
 * Author: stahlhut
 * Created: January 10, 2012
 ********************************************************************
 * Constants of library WL_UserLib
 ********************************************************************)
VAR CONSTANT
	HLKANLINK_MAX_CLIENTCONNS : UINT := 10; (*Anzahl der Clienten *)
	HLKANLINK_MAX_SERVERCONNS : UINT := 10; (*Anzahl der Server *)
	HLKANLINK_MAX_OVERVIEW_DATA : UINT := 31; (*Maximum data transfer on 1 overview connections*)
END_VAR
```

### Package Logical/KanLink_A19/KGFrameworkShare/Pkg_mnTestUser - Testadapter für automatische Test

- Library Logical/KanLink_A19/KGFrameworkShare/Pkg_mnTestUser/libTestUse (IEC) - Userlibrary für Testadapter (no source held here)

### Program Logical/KanLink_A19/KGFrameworkShare/Pkg_mnTestUser/mnTestUser (IEC) - Initialisierung des Test

- KanLink Release Notes.docx (binary file, 15624 bytes)
### Package Logical/KanLink_A19/Examples - * Example Programs

### Program Logical/KanLink_A19/Examples/x_dc1 (IEC, version 1.10.0) - *Discharger with Kanlink Batching

#### dc.var
```iecst
VAR
	BatchQty_Remain : UINT;
	BatchSizeSet : UINT;
	BatchValue : UINT;
	BatchWeight : UINT;
	Check : BOOL;
	CloserDown : BOOL;
	CloserDownET : TIME;
	CloserUp : BOOL;
	CloserUpET : TIME;
	CodeStep : BOOL;
	CodeStepPLS : BOOL;
	Count1 : BOOL;
	DischargerEnable : BOOL;
	ExitLoop : BOOL;
	FaultCount : UINT;
	I_3rdBagLongTrip : BOOL;
	I_BagAtBuffer : BOOL;
	I_BagAtDischarger : BOOL;
	I_BagAtEmptyBuffer : BOOL;
	I_BagEmpty : BOOL;
	I_BagReleased : BOOL;
	I_LoadDropped : BOOL;
	I_OpenBag : BOOL;
	I_SSHC1Closed : BOOL;
END_VAR
VAR RETAIN
	LASTSTEP : UINT;
END_VAR
VAR
	LoadDropped : BOOL;
	MatchCat : BOOL;
	MatchCus : BOOL;
	MinOpen : BOOL;
	MinOpenET : TIME;
	myBag : UINT;
	myBagCloser : BOOL;
	myBuffBag : UINT;
	myCodesStrobe : BOOL;
	myDC : UINT;
	myDst : USINT;
	myIO : UINT;
	myPickerControl : BOOL;
	myPushButtonControl : BOOL;
	myRelCounter : UINT;
	mySeq : UINT;
	myStartStop : UINT;
	myZone : UINT;
	n : UINT;
	O_BagReady : BOOL;
	O_Closer : BOOL;
	O_EmptyBagBufferOpen : BOOL;
	O_OpenBag : BOOL;
	O_OpenBuffer : BOOL;
	O_OpenStop : BOOL;
	O_Steadys : BOOL;
	OpenBagOK : BOOL;
	PLS : BOOL;
	SettledAtBuffer : BOOL;
	SettledAtBufferET : TIME;
	SettledAtDischarger : BOOL;
	SettledAtDischargerET : TIME;
	Start : BOOL;
	SteadysDown : BOOL;
	SteadysDownET : TIME;
	SteadyUp : BOOL;
	SteadyUpET : TIME;
	STEP : UINT;
	Step1Delay : BOOL;
	Step1DelayET : UDINT;
	Temp_BatchSize : UINT;
	TestDischarger : BOOL;
	TestDrop : BOOL;
	TESTTIM : BOOL;
	Timer : BOOL;
	TimerAlarm : TON_10ms;
	TimerET : TIME;
	UseBatch : BOOL;
	UseBuffer : BOOL;
	UseCounter : BOOL;
	BatchValid : BOOL;
	SearchDepth : UINT;
END_VAR
```

#### dc.ab
```automation-basic
;Standard Discharger Sequence

;--------------------------------------------------------------
;Version 1.00 22/04/2011 D.J. First Issue
;Version 1.10 16/08/2011 D.J. Change CodeStep to 4-6 for PT JET
;--------------------------------------------------------------

;Note: the CAN DataType is used for all washing machine interface types CAN bus, BCD / Binary digital and Strobing data.

PROGRAM _CYCLIC

;Configuration
myIO					= 153 	;Discharger IO module number
myStartStop				= 8		;Start / Stop used on TrackView display (Traffic Light)
mySeq					= 8		;Sequence number
myDC					= 3		;Discharger number
myBuffBag				= 376	;Buffer bag number - set to 0 to use Request / Enable
myBag					= 375	;Discharger bag number
myDst					= 33	;Destination number for bags to be opened at this discharger (destination 0 will also be opened)
myRelCounter			= 0 	;Bag released counter number - set to 0 to use RequestRel / EnableRel
myZone					= 0
myBagCloser				= TRUE	;Bag closer is fitted?
myCodesStrobe			= FALSE ;Use Jensen (Senking) strobe method for transfer of codes to CBW
myPushButtonControl		= FALSE ;Bag is opened by pressing a pushbutton and confirmed empty with a second press.
myPickerControl			= FALSE	;Bag is opened by a picker (only open bag signal which goes off when load has dropped
IF myPushButtonControl OR myPickerControl THEN
	CAN[myDC].DropLoad		= X[0].X01 ;Input to open bag?
ENDIF

;Single bag buffer after discharger - enter input and output for the proximity switch and buffer stop.
I_BagAtEmptyBuffer		= FALSE
O_EmptyBagBufferOpen	= FALSE

;/Configuration

DischargerEnable 		= ((D[myStartStop] > 0) AND NOT Std.HaltSysZone[myZone])

I_BagAtBuffer			= X[myIO].X01
I_BagAtDischarger		= X[myIO].X02
I_OpenBag				= CAN[myDC].DropLoad
I_LoadDropped			= CAN[myDC].LoadDropped
;I_BagReleased			= X[myIO].X03
I_BagEmpty			  	= TRUE

O_BagReady				= FALSE
O_OpenBuffer 			= FALSE
O_Steadys				= FALSE
O_Closer				= FALSE
O_OpenBag				= FALSE
O_OpenStop				= FALSE

Request.DC[myDC]		= FALSE
RequestRel.DC[myDC] 	= FALSE

;Alarm
Alarm[mySeq].Name 		= almNoAlarm ;Clear sequence alarm name
Alarm[mySeq].Bag 		= myBag
Alarm[mySeq].Beacon		= TRUE
Alarm[mySeq].Extra		= 0
Alarm[mySeq].Time		= 3000

;Setup Sequence
STEP = D[900 + mySeq]
;Setup Pulse contact
PLS = (STEP <> LASTSTEP)
LASTSTEP = STEP

;Step 0 - Disabled
IF (STEP = 0) THEN
	;Disabled
ENDIF
;*************************************************Batch Calculation**************************************************************
BatchSizeSet	= D[2800 + Bag[myBuffBag].Prg]
BatchQty_Remain = 980 ; D Registers.
BatchWeight 	= 981
MatchCus 		= TRUE

;Calculate buffer data to send to PT - note even 2nd bag of batch will have different weight.
IF (STEP = 1) AND (BatchSizeSet > 1) AND (Bag[myBuffBag].Cat > 0) THEN
	LOOP n = 0 TO 5 DO
		CAN[myDC].Batchpart[n].Customer = 0
		CAN[myDC].Batchpart[n].Wgt = 0
	ENDLOOP
	D[BatchWeight] = Bag[myBuffBag].Wgt
	CAN[myDC].Batchpart[0].Customer = Bag[myBuffBag].Cus
	CAN[myDC].Batchpart[0].Wgt = Bag[myBuffBag].Wgt
	Temp_BatchSize = 1
	ExitLoop = FALSE

	IF (D[BatchQty_Remain] < 1) THEN
		BatchValue = BatchSizeSet
	ELSE
		BatchValue	= D[BatchQty_Remain]
	ENDIF
	IF (BatchValue > 1) THEN
		SearchDepth = 0
		LOOP n = 1 TO (BatchValue - 1)DO
			IF (Bag[myBuffBag + n].Cat > 0) THEN
				SearchDepth = n + 1 ; Add 1 to allow for position 0
			ENDIF
			IF ((Bag[myBuffBag + n].Cat = Bag[myBuffBag].Cat) AND ((Bag[myBuffBag + n].Cus = Bag[myBuffBag].Cus) OR NOT MatchCus))THEN
				D[BatchWeight] = D[BatchWeight] + Bag[myBuffBag + n].Wgt ; Sum Wieghts
				CAN[myDC].Batchpart[n].Customer = Bag[myBuffBag + n].Cus
				CAN[myDC].Batchpart[n].Wgt = Bag[myBuffBag + n].Wgt
				Temp_BatchSize = n + 1
			ELSE
				ExitLoop = TRUE
			ENDIF
		EXITIF ExitLoop
		ENDLOOP
		IF (D[BatchQty_Remain] = 0) AND ((Temp_BatchSize = BatchSizeSet) OR (SearchDepth >= BatchSizeSet)) THEN	; Check we have searched all bags required.
			D[BatchQty_Remain] = Temp_BatchSize
		ENDIF
	ENDIF
ELSE IF (STEP = 1) AND (BatchSizeSet <= 1) AND (Bag[myBuffBag].Cat > 0) THEN
	D[BatchQty_Remain] = 1
	D[BatchWeight] = Bag[myBuffBag].Wgt
	CAN[myDC].Batchpart[0].Customer = Bag[myBuffBag].Cus
	CAN[myDC].Batchpart[0].Wgt = Bag[myBuffBag].Wgt
ENDIF

CAN[myDC].Batch_QtyRemaining = D[BatchQty_Remain]
;*******************************************************END BATCHING CALC****** SEE step 6 from Batch decrement**********************************

;Check Status - Bag settled at buffer, no bag at discharger, bag at buffer on screen and no bag at discharger on the screen
UseBuffer = (myBuffBag > 0)
TON_10ms(I_BagAtBuffer,300,SettledAtBuffer,SettledAtBufferET)
IF (STEP = 1) THEN
	;Disable sequence if input made
	IF (DischargerEnable AND NOT I_BagAtDischarger AND (Bag[myBag].Cat = 0) AND NOT Std.HaltSysZone[myZone]) THEN
		IF UseBuffer THEN
			IF (SettledAtBuffer AND (Bag[myBuffBag].Cat > 0) AND (D[BatchQty_Remain] > 0)) THEN ; Make sure batch size has arrived in buffer.
				D[900 + mySeq] = 2
				INC Count[mySeq]
			ENDIF

			;Alarm - Buffer bag detection error
			IF (Bag[myBuffBag].Cat > 0) AND NOT I_BagAtBuffer THEN
				Alarm[mySeq].Name 	= almBagNotAtProx
				Alarm[mySeq].Bag	= myBuffBag
			ELSE IF (Bag[myBuffBag].Cat = 0) AND I_BagAtBuffer THEN
				Alarm[mySeq].Name 	= almBagNotShownOnScreen
				Alarm[mySeq].Bag	= myBuffBag
			ENDIF

		ELSE
			D[900 + mySeq] = 2
			INC Count[mySeq]
		ENDIF
	ENDIF

	;Alarm - Bag detected at discharger
	IF (Bag[myBag].Cat > 0) THEN
		Alarm[mySeq].Name = almBagDataError
	ELSE IF I_BagAtDischarger THEN
		Alarm[mySeq].Name = almSwitchFault
	ENDIF

ENDIF

;Wait for bag in discharger
IF (STEP = 2) THEN
	O_OpenBuffer 		= UseBuffer
	Request.DC[myDC] 	= NOT UseBuffer
	IF I_BagAtDischarger THEN
		D[900 + mySeq] = 3
	ENDIF
	IF UseBuffer THEN
		Alarm[mySeq].Name = almBagNotArrived
	ENDIF
ENDIF

;Let bag settle in discharger
TON_10ms(I_BagAtDischarger,300,SettledAtDischarger,SettledAtDischargerET)
IF (STEP = 3) THEN
	IF UseBuffer THEN
		IF ((Bag[myBag].Cat = 0) AND (Bag[myBuffBag].Cat > 0)) THEN
			Bag[myBag] 		= Bag[myBuffBag]
			Bag[myBuffBag] 	= Bag[0]
		ENDIF
	ENDIF
	IF ((Bag[myBag].Dst <> myDst) AND (Bag[myBag].Dst <> 0)) THEN
		D[900 + mySeq] = 11 ;Bag is for another destination then go-to release bag
	ENDIF
	IF SettledAtDischarger THEN
		D[900 + mySeq] = 4
	ENDIF
	Alarm[mySeq].Name = almBagNotSettled
ENDIF

;Allow steadys to move down
TON_10ms((STEP = 4),400,SteadysDown,SteadysDownET)
IF (STEP = 4) THEN
	IF SteadysDown AND NOT I_SSHC1Closed THEN
		IF (Bag[myBag].Prg = Std.MaxProg) THEN
			D[900 + mySeq] = 8 ;Empty bag then go-to close
		ELSE
			IF myCodesStrobe THEN
				IF CAN[myDC].StrobeComplete THEN
					D[900 + mySeq] = 5
				ENDIF
			ELSE IF myPushButtonControl THEN
				IF NOT I_OpenBag THEN
					D[900 + mySeq] = 5
				ENDIF
				Alarm[mySeq].Name = almSwitchFault
			ELSE
				D[900 + mySeq] = 5
			ENDIF
		ENDIF
	ENDIF
ENDIF

;Steady cylinders on from steps 4 - 9
O_Steadys = ((STEP >= 4) AND (STEP <= 9))

;Bag opener on from step 5 - 8
O_OpenBag = ((STEP >= 6) AND (STEP <= 8))

CodeStep  = ((STEP >= 5) AND (STEP <= 6))

;Wash Codes

IF CodeStep THEN
	CAN[myDC].Program		= Bag[myBag].Prg
	CAN[myDC].Category 		= Bag[myBag].Cat
	CAN[myDC].Customer 		= Bag[myBag].Cus
	CAN[myDC].Weight   		= D[BatchWeight];Bag[myBag].Wgt  ;(WgtRound / 10) ;rounded up weight divide by 10
	CAN[myDC].BatchID		= Bag[myBag].Mis
	CAN[myDC].DoubleLoad 	= FALSE
ELSE
	CAN[myDC].Program 		= 0
	CAN[myDC].Category 		= 0
	CAN[myDC].Customer 		= 0
	CAN[myDC].Weight   		= 0
	CAN[myDC].BatchID		= 0
	CAN[myDC].DoubleLoad 	= FALSE
ENDIF

;Bag Ready to Washing Machine
IF (STEP = 5) THEN
	;O_BagReady 			= TRUE
	CAN[myDC].BagReady 	= NOT I_SSHC1Closed
	IF I_OpenBag OR TestDischarger THEN
		D[900 + mySeq] = 6
	ENDIF
ELSE
	CAN[myDC].BagReady	= FALSE
ENDIF

;Set LoadDropped to False
IF (STEP <> 6) THEN
	LoadDropped = FALSE
ENDIF

;Open Bag Until LoadDropped Received and has been open for 6 seconds
TON_10ms((STEP = 6),600,MinOpen,MinOpenET) ;ET means Elapsed Time
IF (STEP = 6) THEN

	IF (myPushButtonControl OR myPickerControl) THEN
		IF (NOT I_OpenBag OR TestDischarger) THEN
			LoadDropped = TRUE
		ENDIF
	ELSE
		IF (I_LoadDropped OR TestDischarger) THEN
			LoadDropped = TRUE
		ENDIF
	ENDIF

	IF (LoadDropped AND MinOpen) THEN
		;Write Report
		;------------
		IF (ReportUnloading[myDC].Cat = 0) THEN
			ReportUnloading[myDC].Prg = Bag[myBag].Prg 		;Program
			ReportUnloading[myDC].Cat = Bag[myBag].Cat		;Category
			ReportUnloading[myDC].Cus = Bag[myBag].Cus		;Customer
			ReportUnloading[myDC].Wgt = Bag[myBag].Wgt		;Weight
			ReportUnloading[myDC].Cnt = 0					;Count
			ReportUnloading[myDC].Stn = 0					;Station
			ReportUnloading[myDC].Mcn = myDC				;Machine
			ReportUnloading[myDC].Mis = Bag[myBag].Mis		;Batch ID
			D[BatchQty_Remain] = (D[BatchQty_Remain] - 1)
			D[900 + mySeq] = 7
		ENDIF
	Alarm[mySeq].Time = 60000
	Alarm[mySeq].Name = almLoadNotDropped
	ENDIF
ENDIF
;Change display to empty bag - clear all other bag data
IF (STEP = 7) THEN
	IF myPushButtonControl THEN
		O_BagReady 	= Std.Clock200ms
		IF ((I_OpenBag AND NOT I_LoadDropped AND I_BagEmpty) OR TestDrop) THEN
			Bag[myBag]		= Bag[0]
			Bag[myBag].Prg 	= Std.MaxProg
			Bag[myBag].Cat	= Std.MaxCats
			D[900 + mySeq] 		= 8
		ENDIF
		IF (I_LoadDropped OR I_BagEmpty) THEN
			Alarm[mySeq].Name = almSwitchFault
		ENDIF
	ELSE
		IF ((NOT I_OpenBag AND NOT I_LoadDropped AND I_BagEmpty) OR TestDrop) THEN
			Bag[myBag]		= Bag[0]
			Bag[myBag].Prg 	= Std.MaxProg
			Bag[myBag].Cat	= Std.MaxCats
			D[900 + mySeq] 		= 8
		ENDIF
		IF (I_OpenBag OR I_LoadDropped OR I_BagEmpty) THEN
			Alarm[mySeq].Name = almSwitchFault
		ENDIF
	ENDIF
ENDIF

;Close bag
TON_10ms((STEP = 8),700,CloserDown,CloserDownET)
IF (STEP = 8) THEN
	IF myBagCloser THEN
		O_Closer = TRUE
		IF CloserDown THEN
			D[900 + mySeq] = 9
		ENDIF
	ELSE
		D[900 + mySeq] = 10
	ENDIF
ENDIF

;Allow closer to go back up
TON_10ms((STEP = 9),700,CloserUp,CloserUpET)
IF (STEP = 9) THEN
	IF CloserUp THEN
		D[900 + mySeq] = 10
	ENDIF
ENDIF

;Allow steadys to go up
TON_10ms((STEP = 10),400,SteadyUp,SteadyUpET)
IF (STEP = 10) THEN
	IF SteadyUp AND NOT EnableRel.DC[myDC] THEN
		D[900 + mySeq] = 11
	ENDIF
ENDIF

;Check for space on empty bag buffer / Request release
UseCounter = (myRelCounter > 0)
IF (STEP = 11) THEN
	IF UseCounter THEN
		IF (Line[myRelCounter].Clear AND NOT I_BagAtEmptyBuffer AND NOT O_EmptyBagBufferOpen) THEN
			D[900 + mySeq] = 12
		ENDIF
		IF (Line[myRelCounter].Clear AND I_BagAtEmptyBuffer AND NOT O_EmptyBagBufferOpen) THEN
			Alarm[mySeq].Name = almSwitchFault
		ENDIF
	ELSE
		RequestRel.DC[myDC]	= TRUE
		IF EnableRel.DC[myDC] THEN
			D[900 + mySeq] = 12
		ENDIF
	ENDIF
ENDIF

;Open buffer stop - unitl bag out
IF (STEP = 12) THEN
	O_OpenStop = TRUE
	Bag[myBag] = Bag[0] ;Clear bag

	IF UseCounter THEN
		IF PLS THEN
			C[myRelCounter] = 0
		ENDIF
		IF Line[myRelCounter].Trip OR I_BagReleased THEN
			D[900 + mySeq] = 1
		ENDIF
	ELSE
		IF NOT EnableRel.DC[myDC] THEN
			D[900 + mySeq] = 1
		ENDIF
	ENDIF
	Alarm[mySeq].Name = almBagNotReleased
ENDIF

;*************************************************

;Alarms
TimerAlarm.IN 	= NOT PLS AND (Alarm[mySeq].Name > 0)
TimerAlarm.PT 	= Alarm[mySeq].Time
TimerAlarm FUB TON_10ms()
Alarm[mySeq].On 	= TimerAlarm.Q
Alarm[mySeq].ET 	= TimerAlarm.ET

;Outputs
;Y[24].Y16 		= O_BagReady
Y[myIO].Y04 	= O_OpenBuffer
Y[myIO].Y05 	= O_Steadys
Y[myIO].Y06 	= O_OpenBag
Y[myIO].Y07 	= O_Closer
Y[myIO].Y08 	= O_OpenStop

END_PROGRAM
```

- Visualisation Logical/Displays/PCT04 (not shown)

- Visualisation Logical/Displays/CT11 (not shown)

### DisplaysGlobal.typ - Global Datatype
```iecst
(********************************************************************
 * COPYRIGHT -- Bernecker + Rainer
 ********************************************************************
 * Package: LibAsTCP
 * File: LibAsTCP.typ
 * Author: Bernecker + Rainer
 * Created: February 21, 2008
 ********************************************************************
 * Data types of package LibAsTCP
 ********************************************************************)

TYPE
	myPanel_typ : 	STRUCT
		Text : STRING[20];
		Datapoint : DINT;
		Min : DINT;
		Max : DINT;
		Status : UINT;
		Completion : UINT;
		Locking : UINT;
	END_STRUCT;
	pnlDisplay_Typ : 	STRUCT
		ClientIP : STRING[16]; (*Connectec Client IP Address*)
		SendData : ARRAY[0..3]OF pnlDisplaySend_Typ; (*Send Data*)
		ReceiveData : ARRAY[0..3]OF pnlDisplayReceive_Typ; (*Reveive Data*)
	END_STRUCT;
	pnlDisplayReceive_Typ : 	STRUCT
		Language : UINT; (*Language selection*)
		Command : UINT; (*Command Received from panel eg. Button Pressed*)
		DataEntry1 : UDINT; (*Data entry value*)
		DataEntry2 : UDINT; (*Data entry value*)
		DataEntry3 : UDINT; (*Data entry value*)
		DataEntry4 : UDINT; (*Data entry value*)
		DataEntry5 : UDINT; (*Data entry value*)
		DataEntry6 : UDINT; (*Data entry value*)
	END_STRUCT;
	pnlDisplaySend_Typ : 	STRUCT
		Language : USINT; (*Language from Master PLC*)
		IP_Address : STRING[16]; (*New Display IP Address the Gateway takes the complete address the IP and Server only the first 3 parts*)
		CycleSync_ms : UINT; (*Server sync cycle time*)
		SYSreset : UINT; (*System Reset (cold start etc..)*)
		Brightness : UINT; (*Panel Brightness*)
		MainDisplay : UINT; (*Selection of various main displays set from 20 onwards*)
		MainColour : UINT; (*Main foreground and background colour*)
		DisplayBag : Bag_typ; (*Display data for bag text*)
		TextColour1 : UINT; (*Text foreground and background colour*)
		TextColour2 : UINT; (*Text foreground and background colour*)
		TextColour3 : UINT; (*Text foreground and background colour*)
		TextColour4 : UINT; (*Text foreground and background colour*)
		TextColour5 : UINT; (*Text foreground and background colour*)
		TextColour6 : UINT; (*Text foreground and background colour*)
		Max1 : UDINT; (*Data entry limit*)
		Max2 : UDINT; (*Data entry limit*)
		Max3 : UDINT; (*Data entry limit*)
		Max4 : UDINT; (*Data entry limit*)
		Max5 : UDINT; (*Data entry limit*)
		Max6 : UDINT; (*Data entry limit*)
		SQL : SQLLogin_typ;
		StnName : STRING[5];
		CustomText : ARRAY[0..4]OF STRING[25];
	END_STRUCT;
	pnlClient_Typ : 	STRUCT
		ButtonPressed : UINT;
		CurrentPage : UINT;
		ChangePage : UINT;
		IFport : STRING[16];
		ServerIPaddress : STRING[16];
		IPaddress : STRING[16];
		SubnetMask : STRING[16];
		Gateway : STRING[16];
		BroadcastAddress : STRING[16];
		Password : UINT;
		ServerCycle_ms : UINT;
	END_STRUCT;
	pnlTextType : 	STRUCT
		Prg : UDINT;
		PrgLong : STRING[8];
		PrgName : STRING[50];
		Cat : UDINT;
		CatLong : STRING[8];
		CatName : STRING[50];
		Cus : UDINT;
		CusLong : STRING[8];
		CusName : STRING[50];
		ImagePath : STRING[32];
		Description : STRING[10];
	END_STRUCT;
END_TYPE
```

### DisplaysGlobal.var - Data for AsTCP Global Variables
```iecst
(********************************************************************
 * COPYRIGHT -- Bernecker + Rainer
 ********************************************************************
 * Package: LibAsTCP
 * File: LibAsTCP.var
 * Author: Bernecker + Rainer
 * Created: February 21, 2008
 ********************************************************************
 * Variables of package LibAsTCP
 ********************************************************************)
VAR
	ClientText : ARRAY[0..3] OF pnlTextType;
END_VAR
VAR RETAIN
	ClientServerIP : STRING[16];
END_VAR
VAR
	ClientGeneral : pnlClient_Typ;
	ClientReceive : ARRAY[0..3] OF pnlDisplaySend_Typ; (*Single Dimension Receive Array for Client Panel*)
	ClientSend : ARRAY[0..3] OF pnlDisplayReceive_Typ; (*Single Dimension Send Array for Client Panel*)
	DisplayData : ARRAY[0..19] OF pnlDisplay_Typ;
END_VAR
```

### Program Logical/Displays/ServerPanel (IEC, version 4.00.0) - Server Build Panel Data

#### ServerPanel.ab - Implementation code
```automation-basic
(********************************************************************
 * COPYRIGHT --
 ********************************************************************
 * Program: DisplayBuild
 * File: DisplayBuild.ab
 * Author: Dave
 * Created: December 08, 2010
 ********************************************************************
 * Implementation of program Server Panel
 ********************************************************************)

;Version 1.00 12/12/2010 D.J. First Issue
;Version 2.00 30/06/2011 D.J. Changed weight value to INT to display minus numbers
;Version 3.00 20/07/2011 D.J. Added Code for CTT11 4 Displays on 1 screen (Quadrants)
;Version 4.00 18/10/2011 D.J. Added Data Entry Panel

PROGRAM _INIT

    ;Each Display Can send and receive upto 4 sets of data then Node is used to control which is sent
	;All displays should get their names using the zzGetNames function including Data Entry panels which should have a panel bag as before.

	;Set Display indemyNode
	DisplayDataSize = (SIZEOF(DisplayData) / SIZEOF(DisplayData[0])) - 1
	NodeDataSize 	= (SIZEOF(NodeData) / SIZEOF(NodeData[0])) - 1

	;Foreground and Background colours
	BgBlack 	= $0000
	BgBlue		= $0001
	BgLtBlue	= $0009
	BgWhite		= $000F
	BgRed		= $0033
	BgOrange	= $002A
	BgLtGray	= $0007
	BgGray		= $0008

	FgBlack		= $0000
	FgBlue		= $0100
	FgLtBlue	= $0900
	FgWhite		= $0F00
	FgRed		= $3300
	FgOrange	= $2A00
	FgLtGray	= $0700
	FgGray		= $0800

	myDisplay 	= TypeDataEntry	;Set to required main display 0 = Default
	mySyncTime	= 100 	;100ms Default
	NodeOffset 	= 31	;First Display Node

	LOOP myNode = 1 TO 2 DO
		NodeData[myNode].DsplayType = TypeDataEntry
	ENDLOOP
   LOOP myNode = 3 TO 4 DO
		NodeData[myNode].DsplayType = TypeDisplay
		IF myNode = 3 THEN
			strcpy(ADR(NodeData[myNode].Quadrant[myQuad].StnName),"SVC1")
		ELSE IF myNode = 4 THEN
			strcpy(ADR(NodeData[myNode].Quadrant[myQuad].StnName),"SVC2")
		ENDIF
	ENDLOOP
	;Setup each Display Node
	LOOP myNode = 1 TO NodeDataSize DO
		IF NodeData[myNode].DsplayType = TypeDisplay THEN

			NodeData[myNode].MainDisplay = 21

			NodeData[myNode].MainColour	= (BgWhite + FgBlue)
			LOOP myQuad = 0 TO 3 DO
				itoa(stnIndex,ADR(myStnString))

				INC stnIndex
				;strcpy(ADR(NodeData[myNode].Quadrant[myQuad].StnName),"SSK1")
				NodeData[myNode].Quadrant[myQuad].TextColour1 	= (BgOrange + FgBlue) ;(BgLtBlue + FgWhite)
				NodeData[myNode].Quadrant[myQuad].TextColour2 	= (BgWhite + FgBlue)
				NodeData[myNode].Quadrant[myQuad].TextColour3 	= (BgWhite + FgBlue)
				NodeData[myNode].Quadrant[myQuad].TextColour4 	= (BgWhite + FgBlue)
				NodeData[myNode].Quadrant[myQuad].TextColour5 	= (BgBlue  + FgWhite)
;				NodeData[myNode].Quadrant[myQuad].TextColour6 	= (BgWhite + FgBlue)
			ENDLOOP

		ELSE IF NodeData[myNode].DsplayType = TypeDataEntry THEN
			itoa(stnIndex,ADR(myStnString))
			strcpy(ADR(NodeData[myNode].Quadrant[0].StnName),ADR(myStnString))
			NodeData[myNode].MainDisplay = 201
			NodeData[myNode].MainColour	= (BgRed + BgWhite)
			LOOP myQuad = 0 TO 3 DO
				NodeData[myNode].Quadrant[myQuad].TextColour1 	= (BgRed + FgRed) ;(BgLtBlue + FgWhite)
				NodeData[myNode].Quadrant[myQuad].TextColour2 	= (BgRed + FgRed)
				NodeData[myNode].Quadrant[myQuad].TextColour3 	= (BgRed + FgRed)
				NodeData[myNode].Quadrant[myQuad].TextColour4 	= (BgRed + FgRed)
				NodeData[myNode].Quadrant[myQuad].TextColour5 	= (BgRed + FgRed)
				NodeData[myNode].Quadrant[myQuad].TextColour6 	= (BgRed + FgRed)

				NodeData[myNode].Quadrant[myQuad].Max1 			= Std.MaxProg ;Program not entered
				NodeData[myNode].Quadrant[myQuad].Max2 			= Std.MaxCats	;Cats
				NodeData[myNode].Quadrant[myQuad].Max3 			= Std.MaxCust	;Customers
				NodeData[myNode].Quadrant[myQuad].Max4 			= Std.MaxLines ; Destination
				NodeData[myNode].Quadrant[myQuad].Max5 			= 0	;Not Used
				NodeData[myNode].Quadrant[myQuad].Max6 			= 0	;Not Used
			ENDLOOP
		ENDIF
	ENDLOOP

	;Setup the BagIndex for each Node and Sub Quadrant	- PCT 03 Would Normally Only Use Quadrant 0
	LOOP n = 1 TO 2 DO
		NodeData[n].Quadrant[0].BagIndex = 310
	;	NodeData[n].Quadrant[1].BagIndex = 0
	;	NodeData[n].Quadrant[2].BagIndex = 0
	;	NodeData[n].Quadrant[3].BagIndex = 0
	ENDLOOP
	LOOP n = 3 TO 4 DO
		NodeData[n].Quadrant[0].BagIndex = 100 + n
	;	NodeData[n].Quadrant[1].BagIndex = 0
	;	NodeData[n].Quadrant[2].BagIndex = 0
	;	NodeData[n].Quadrant[3].BagIndex = 0
	ENDLOOP

	strcpy(ADR(pnlStatusString[0]),ADR("1"))
	strcpy(ADR(pnlStatusString[1]),ADR("Invalid Read"))
	strcpy(ADR(pnlStatusString[2]),ADR("Enter Bag Number"))
	strcpy(ADR(pnlStatusString[3]),ADR("Please Wait"))
	strcpy(ADR(pnlStatusString[4]),ADR(""))
;	strcpy(ADR(pnlStatusString[5]),ADR("No bag on carriage"))
;	strcpy(ADR(pnlStatusString[6]),ADR("Weight not valid"))
;	strcpy(ADR(pnlStatusString[7]),ADR("Program not valid"))

END_PROGRAM

PROGRAM _CYCLIC

	ScreenSave  = 0
	Connected = FALSE
	TON_10ms(ScreenSave,3000,BacklightOff,BackLightOffET)

	LOOP myConn = 0 TO UINT(DisplayDataSize) DO

		;Check if connected - Client IP address
		Status 		= ethInetAton(ADR(DisplayData[myConn].ClientIP),ADR(ClientIP))
		ClientNode 	= 0
		IF Status = 0 THEN
			;Get the connected node number from the IP address
			Node 		= swapUDINT(ClientIP) ;Mask out the IP address
			ClientNode 	= (Node AND $000000FF)
		ENDIF

		IF (ClientNode > 0) THEN

			;Node to Display Number (myNode)
			myNode = 0 ;Default Send zzGetNamesData[0] / Unknown display connected
			IF ((ClientNode >= 31) AND (ClientNode <= 47)) THEN
				myNode = (ClientNode - (NodeOffset - 1))
			ENDIF

			DisplayData[myConn].SendData[0].SQL = SQL.Login
			DisplayData[myConn].SendData[0].MainColour 		= NodeData[myNode].MainColour
			DisplayData[myConn].SendData[0].CycleSync_ms 	= mySyncTime
			DisplayData[myConn].SendData[0].MainDisplay 	= NodeData[myNode].MainDisplay

			DisplayData[myConn].SendData[0].Max1 			= Std.MaxProg ;Program not entered
				DisplayData[myConn].SendData[0].Max2 			= Std.MaxCats	;Cats
				DisplayData[myConn].SendData[0].Max3 			= Std.MaxCust	;Customers
				DisplayData[myConn].SendData[0].Max4 			= Std.MaxLines

			IF BacklightOff THEN
				DisplayData[myConn].SendData[0].Brightness = 0 ;0 Will also turn off the backlight
			ELSE IF ScreenSave THEN
				DisplayData[myConn].SendData[0].Brightness = 1 ;0 Will also turn off the backlight
			ELSE
				DisplayData[myConn].SendData[0].Brightness = 100
			ENDIF

			LOOP myQuad = 0 TO 3 DO

				IF myNode < 10 THEN
				;	itoa(NodeData[myNode].Quadrant[myQuad].BagIndex - (Std.StationBagDisplay[1] - 1) ,ADR(NodeData[myNode].Quadrant[myQuad].StnName))
				ELSE
					strcpy(ADR(NodeData[myNode].Quadrant[myQuad].StnName),"SSK1")
				ENDIF
				strcpy(ADR(DisplayData[myConn].SendData[myQuad].StnName),ADR(NodeData[myNode].Quadrant[myQuad].StnName))
				myBag	= NodeData[myNode].Quadrant[myQuad].BagIndex

				IF (myBag > 0) THEN

                  DisplayData[myConn].SendData[myQuad].DisplayBag = Bag[myBag]

					strcpy(ADR(myMessageString),"SP2= ")
					mySP = D32[104]
					mySP = mySP/10
					length = ftoa(mySP,ADR(mySPString))
					next_adr = strcat(ADR(myMessageString),ADR(mySPString))
					next_adr = strcat(ADR(myMessageString)," Kg")

					strcpy(ADR(DisplayData[myConn].SendData[myQuad].CustomText[0]),ADR(myMessageString))
					IF Bag[99].Wgt > D32[105] THEN
						strcpy(ADR(myMessageString),"SP3= ")
						mySP = D32[105]
						mySP = mySP/10
						length = ftoa(mySP,ADR(mySPString))
						next_adr = strcat(ADR(myMessageString),ADR(mySPString))
						next_adr = strcat(ADR(myMessageString)," Kg")

						strcpy(ADR(DisplayData[myConn].SendData[myQuad].CustomText[0]),ADR(myMessageString))
						IF NOT Std.Clock1s THEN
							DisplayData[myConn].SendData[myQuad].TextColour6 = (BgRed + FgBlue); (FgRed + BgWhite)
						ELSE
							DisplayData[myConn].SendData[myQuad].TextColour6 =  (FgRed + BgWhite)
						ENDIF
					ELSE IF Bag[201].Wgt < D32[104] THEN
 						DisplayData[myConn].SendData[myQuad].TextColour6 = (BgWhite + FgBlue)
					ELSE IF Bag[99].Wgt > D32[104] THEN
						strcpy(ADR(myMessageString),"SP2= ")
						mySP = D32[104]
						mySP = mySP/10
						length = ftoa(mySP,ADR(mySPString))
						next_adr = strcat(ADR(myMessageString),ADR(mySPString))
						next_adr = strcat(ADR(myMessageString)," Kg")
						strcpy(ADR(DisplayData[myConn].SendData[myQuad].CustomText[0]),ADR(myMessageString))
						;IF NOT Std.Clock1s THEN
							DisplayData[myConn].SendData[myQuad].TextColour6 = (BgRed + FgBlue); (FgRed + BgWhite)
						;ELSE
						;	DisplayData[myConn].SendData[myQuad].TextColour6 =  (FgRed + BgWhite)
						;ENDIF
;						DisplayData[myConn].SendData[myQuad].TextColour5 = (BgRed + FgRed)
;						DisplayData[myConn].SendData[myQuad].TextColour4 = (BgRed + FgRed)
;						DisplayData[myConn].SendData[myQuad].TextColour3 = (BgRed + FgRed)
;						DisplayData[myConn].SendData[myQuad].TextColour2 = (BgRed + FgRed)
;						DisplayData[myConn].SendData[myQuad].TextColour1 = (BgRed + FgRed)
					ENDIF

;					IF (myBag > 200) THEN
;						StnNo = (myBag - 200)
;					ENDIF
;					IF Y[300 + StnNo].Y07 THEN
;						NodeData[myNode].Quadrant[myQuad].Max1 			= Std.MaxProg ;Program not entered
					;	NodeData[myNode].Quadrant[myQuad].Max2 			= Std.MaxCats	;Cats
					;	NodeData[myNode].Quadrant[myQuad].Max3 			= Std.MaxCust	;Customers
					;	NodeData[myNode].Quadrant[myQuad].Max4 			= Std.MaxLines ; Destination
;					ELSE
						DisplayData[myConn].SendData[myQuad].TextColour1 	= (BgOrange + FgRed) ;Customer
						DisplayData[myConn].SendData[myQuad].TextColour2 	= (BgWhite + FgRed) ; Cat Long
						DisplayData[myConn].SendData[myQuad].TextColour3 	= (BgWhite + FgRed); Cat
						DisplayData[myConn].SendData[myQuad].TextColour4 	= (BgWhite + FgRed) ; Count
						DisplayData[myConn].SendData[myQuad].TextColour5 	= (BgWhite + FgRed) ; Wieght
	;					DisplayData[myConn].SendData[myQuad].TextColour6 	= (BgWhite + FgBlue) ; Stn
;					ENDIF

					;Copy Data Entry to Local
					NodeData[myNode].Quadrant[myQuad].DataEntry1 			= DisplayData[myConn].ReceiveData[myQuad].DataEntry1
					NodeData[myNode].Quadrant[myQuad].DataEntry2 			= DisplayData[myConn].ReceiveData[myQuad].DataEntry2
					NodeData[myNode].Quadrant[myQuad].DataEntry3 			= DisplayData[myConn].ReceiveData[myQuad].DataEntry3
					NodeData[myNode].Quadrant[myQuad].DataEntry4 			= DisplayData[myConn].ReceiveData[myQuad].DataEntry4
					NodeData[myNode].Quadrant[myQuad].DataEntry5 			= DisplayData[myConn].ReceiveData[myQuad].DataEntry5
					NodeData[myNode].Quadrant[myQuad].DataEntry6 			= DisplayData[myConn].ReceiveData[myQuad].DataEntry6

					NodeData[myNode].Quadrant[myQuad].Command				= DisplayData[myConn].ReceiveData[myQuad].Command

;					;Copy Entered Data to Bag Data
					IF NodeData[myNode].DsplayType = TypeDataEntry THEN
						Connected = TRUE
					;	Bag[myBag] = DisplayData[myNode].ReceiveData[myQuad].DataEntryBag
						Bag[myBag].Cat = NodeData[myNode].Quadrant[myQuad].DataEntry2
						Bag[myBag].Cus = NodeData[myNode].Quadrant[myQuad].DataEntry3
						Bag[myBag].Dst = USINT(NodeData[myNode].Quadrant[myQuad].DataEntry4)
					;ELSE IF NodeData[myNode].DsplayType = TypeMaintLine THEN
						;zzMaintLine[myNode].Data = UINT(NodeData[myNode].Quadrant[myQuad].DataEntry3)
						ELSE

					ENDIF

				ENDIF ;/myGetIdx > 0
			ENDLOOP ;/myQuad

			;Restart Display
			IF RestartDisplays THEN
				DisplayData[myConn].SendData[0].SYSreset = 1
			ENDIF

		ENDIF

		;Cancel Restart Display
		IF RestartComplete THEN
			DisplayData[myConn].SendData[0].SYSreset = 0
			IF (myConn = DisplayDataSize) THEN
				RestartDisplays	= FALSE 	;Cancel Re-start when last display
			ENDIF
		ENDIF

		;Change IP address
		IF ReplaceIP THEN
			strcpy(ADR(DisplayData[myConn].SendData[0].IP_Address),ADR(ReplaceIPAddress))
		ENDIF

		;Cancel Replace IP
		IF ReplaceIPComplete THEN
			strcpy(ADR(DisplayData[myConn].SendData[0].IP_Address),ADR(""))
			ReplaceIP = FALSE 	;Cancel Replace IP when last display
		ENDIF

	ENDLOOP
	SkipMarker:
	;Cancel re-start timer
	TON_10ms(RestartDisplays,200,RestartComplete,RestartCompleteET)
	TON_10ms(ReplaceIP,200,ReplaceIPComplete,ReplaceIPCompleteET)

;	Y[15].Y15 = NOT Connected
;	CAN[1].Live = NOT Y[5].Y15
END_PROGRAM
```

#### ServerPanel.typ - Local data types
```iecst
(********************************************************************
 * COPYRIGHT --
 ********************************************************************
 * Program: DisplayBuild
 * File: DisplayBuild.typ
 * Author: Dave
 * Created: December 08, 2010
 ********************************************************************
 * Local data types of program DisplayBuild
 ********************************************************************)

TYPE
	pnlNodeData_typ : 	STRUCT
		DsplayType : UINT; (*Display Type ie. 0=Display 1=DataEntry*)
		MainDisplay : UINT; (*Required Main Display Page eg.. 22*)
		MainColour : UINT; (*Main Display Colour*)
		Quadrant : ARRAY[0..3]OF pnlNodeValues_typ;
	END_STRUCT;
	pnlNodeValues_typ : 	STRUCT
		BagIndex : UINT; (*zzGetNamesIndex - *)
		Command : UINT; (*Received Command ie. Start Button Pressed = 1*)
		Description : UINT; (*Station number*)
		DataEntry1 : UDINT; (*Data entry value 1*)
		DataEntry2 : UDINT; (*Data entry value 2*)
		DataEntry3 : UDINT; (*Data entry value 3*)
		DataEntry4 : UDINT; (*Data entry value 4*)
		DataEntry5 : UDINT; (*Data entry value 5*)
		DataEntry6 : UDINT; (*Data entry value 6*)
		TextColour1 : UINT; (*Text 1 foreground and background colour*)
		TextColour2 : UINT; (*Text 2 foreground and background colour*)
		TextColour3 : UINT; (*Text 3 foreground and background colour*)
		TextColour4 : UINT; (*Text 4 foreground and background colour*)
		TextColour5 : UINT; (*Text 5 foreground and background colour*)
		TextColour6 : UINT; (*Text 6 foreground and background colour*)
		Max1 : UDINT; (*Data entry limit 1*)
		Max2 : UDINT; (*Data entry limit 2*)
		Max3 : UDINT; (*Data entry limit 3*)
		Max4 : UDINT; (*Data entry limit 4*)
		Max5 : UDINT; (*Data entry limit 5*)
		Max6 : UDINT; (*Data entry limit 6*)
		StnName : STRING[5];
	END_STRUCT;
END_TYPE
```

#### ServerPanel.var - Local variables
```iecst
(********************************************************************
 * COPYRIGHT --
 ********************************************************************
 * Program: DisplayBuild
 * File: DisplayBuild.var
 * Author: Dave
 * Created: December 08, 2010
 ********************************************************************
 * Local variables of program DisplayBuild
 ********************************************************************)
VAR CONSTANT
	TypeDisplay : UINT := 22;
	TypeDataEntry : UINT := 1;
END_VAR
VAR
	BacklightOff : BOOL;
	BackLightOffET : UDINT;
	BgBlack : UINT;
	BgBlue : UINT;
	BgLtBlue : UINT;
	BgLtGray : UINT;
	BgOrange : UINT;
	BgRed : UINT;
	BgWhite : UINT;
	ClientIP : UDINT;
	ClientNode : UDINT;
	DisplayDataSize : UDINT;
	DisplaySize : UDINT;
	FgBlack : UINT;
	FgBlue : UINT;
	FgLtBlue : UINT;
	FgLtGray : UINT;
	FgOrange : UINT;
	FgRed : UINT;
	FgWhite : UINT;
	length : UINT;
	myBag : UINT;
	myDisplay : UINT;
	mySync : UINT;
	mySyncTime : UINT;
	myTextColour : ARRAY[0..6] OF UINT;
	myWeight : REAL;
	myWeightString : STRING[8];
	n : UINT;
	Node : UDINT;
	NodeOffset : UINT;
	nxt_adr : UDINT;
	RestartComplete : BOOL;
	RestartCompleteET : UDINT;
	RestartDisplays : BOOL;
	ScreenSave : BOOL;
	Status : UINT;
	x : UDINT;
	myCustomerString : STRING[80];
	myProgramString : STRING[80];
	myCategoryString : STRING[80];
	MyNewIP : STRING[16];
	IP_Replace_0 : IP_Replace;
	Dave : BOOL;
	MyReplaceIP : STRING[16];
	ReplaceIPAddress : STRING[16]; (*Actual the new required Gateway the IP and Server will take the first 3 parts and the 4 will be the same.*)
	ReplaceIP : BOOL;
	ReplaceIPComplete : BOOL;
	ReplaceIPCompleteET : UDINT;
	lenght : UINT;
	myINTweight : INT;
	NodeData : ARRAY[0..19] OF pnlNodeData_typ;
	NodeDataSize : UINT;
	ns : UINT;
	myColour : UINT;
	myNode : UDINT;
	myQuad : UINT;
	myGetIdx : UINT;
	myConn : UINT;
	next_adr : UDINT;
	myGetIndexString : STRING[80];
	BgGray : UINT;
	FgGray : UINT;
	pnlStatusString : ARRAY[0..19] OF STRING[25];
	myMessageString : STRING[25];
	myStatusColour : UINT;
	Catlenght : UINT;
	myLength : UINT;
	myCatLength : ARRAY[0..20] OF UINT;
END_VAR
VAR CONSTANT
	TypeDisplayPP65 : UINT := 2;
END_VAR
VAR
	myCountString : STRING[8];
	BgGreen : USINT;
END_VAR
VAR CONSTANT
	TypeDisplayCTT104 : UINT := 3;
	TypeDisplayPP65ES1 : UINT := 4;
END_VAR
VAR
	myCount : UINT;
	Disp : INT;
	TypeMaintLine : UINT;
	myWgt : UINT;
	myBarrowCusString : STRING[80];
	myCDC24CusString : STRING[80];
	myCSB2CatString : STRING[80];
	myCCD2CatString : STRING[80];
	myBarrowCatString : STRING[80];
	myCbs2CusPUString : STRING[80];
	TypeBrolli : BOOL;
	myPictureString : BOOL;
	SP1 : UDINT;
	SP2 : UDINT;
	SP3 : UDINT;
	zzMaintLine : BOOL;
	StnNo : UINT;
	stnIndex : UINT;
	myStnString : STRING[5];
	mySP : UDINT;
	mySPString : STRING[25];
	Connected : BOOL;
END_VAR
```

### Program Logical/Displays/Server (IEC, version 2.00.0) - AsTCP Server Application

#### Server.ab - Implementation code
```automation-basic
(********************************************************************
 * COPYRIGHT --
 ********************************************************************
 * Program: NewProgram
 * File: NewProgram.ab
 * Author: Dave
 * Created: December 01, 2010
 ********************************************************************
 * Implementation of program NewProgram
 ********************************************************************)

;Version 1.00 12/12/2010 D.J. First Issue
;Version 2.00 03/02/2010 D.J. Revised connection close code for each connection - added connection count for fault finding.

PROGRAM _INIT

	ServerSize 		= (SIZEOF(Server) / SIZEOF(Server[0]))
	myMaxConns		= (UINT(ServerSize) - 1)

	LOOP n = 0 TO myMaxConns DO
		Server[n].Status = sckError
	ENDLOOP

	ServerOpen.Status = sckClosed

	IF ((IdentRetain > 0) AND (ServerOpen.TcpOpen_0.ident = 0)) THEN
		ServerOpen.TcpOpen_0.ident = IdentRetain
	ENDIF

END_PROGRAM

PROGRAM _CYCLIC

	;Init Ethernet Socket - Pause after any close etc
	TON_10ms_0.IN = (ServerOpen.Status = sckClosed)
	TON_10ms_0.PT = 100
	TON_10ms_0 FUB TON_10ms()

	IF TON_10ms_0.Q THEN
		ServerOpen.Status = sckConnecting
	ENDIF

	;Open Ethernet Socket
	IF ServerOpen.Status = sckConnecting THEN

		ServerOpen.TcpOpen_0.enable  	= TRUE
		ServerOpen.TcpOpen_0.pIfAddr 	= 0					;  (* Listen on all TCP/IP Interfaces*)
		ServerOpen.TcpOpen_0.port 		= 12000				;  (* Port to listen*)
		ServerOpen.TcpOpen_0.options 	= tcpOPT_REUSEADDR	;
		ServerOpen.TcpOpen_0 FUB TcpOpen() 								;  (* Call the Function*)

		IF ServerOpen.TcpOpen_0.status = 0 THEN  (* TcpOpen successfull*)
			ServerOpen.Status 	= sckSetLinger ;sckConnected
			IdentRetain			= ServerOpen.TcpOpen_0.ident
		ELSE IF ServerOpen.TcpOpen_0.status = ERR_FUB_BUSY THEN  (* TcpOpen not finished -> redo *)
		 	;Busy
		ELSE IF ServerOpen.TcpOpen_0.status = tcpERR_ALREADY_EXIST THEN
			ServerOpen.Status = sckError
		ELSE IF ServerOpen.TcpOpen_0.status = tcpERR_SOCKET_BIND THEN
			ServerOpen.Status = sckError
		ENDIF
	ENDIF

	;Set Open Linger Options
	IF ServerOpen.Status = sckSetLinger THEN

		ServerOpen.linger_opt.lLinger 	= 0 ;Linger Time = 0
		ServerOpen.linger_opt.lOnOff	= 1	;Linger Option On

		ServerOpen.TcpIoctl_0.enable 	= TRUE
		ServerOpen.TcpIoctl_0.ident 	= ServerOpen.TcpOpen_0.ident
		ServerOpen.TcpIoctl_0.ioctl		= tcpSO_LINGER_SET
		ServerOpen.TcpIoctl_0.pData		= ADR(ServerOpen.linger_opt)
		ServerOpen.TcpIoctl_0.datalen 	= SIZEOF(ServerOpen.linger_opt)
		ServerOpen.TcpIoctl_0 FUB TcpIoctl()

		IF ServerOpen.TcpIoctl_0.status = 0 THEN
			ServerOpen.Status = sckConnected
		ELSE IF ServerOpen.TcpIoctl_0.status = ERR_FUB_BUSY THEN  (* TcpIoctl not finished -> redo *)
		 	;Busy
		ENDIF

	ENDIF

	;Close Ethernet Socket
	IF ServerOpen.Status = sckError THEN

		ServerOpen.TcpClose_0.enable 	= TRUE
		ServerOpen.TcpClose_0.ident 	= ServerOpen.TcpOpen_0.ident
		ServerOpen.TcpClose_0.how 		= 0;; // tcpSHUT_RD OR tcpSHUT_WR;
		ServerOpen.TcpClose_0 FUB TcpClose()

		IF ServerOpen.TcpClose_0.status = 0 THEN
			ServerOpen.Status = sckClosed
			LOOP n = 0 TO myMaxConns DO
				Server[n].Status = sckError
			ENDLOOP
		ELSE IF ServerOpen.TcpClose_0.status = ERR_FUB_BUSY THEN  (* TcpClose not finished -> redo *)
		 	;Busy
		ELSE IF ServerOpen.TcpClose_0.status = tcpERR_INVALID_IDENT THEN
			ServerOpen.Status = sckClosed
		ENDIF

	ENDIF

	;Get the IO control status
	IF (ServerOpen.Status <> sckSetLinger) THEN

		IF IoctlStatus = ID_List_get THEN
			;Get list of open idents
			ServerOpen.TcpIoctl_0.enable 	= TRUE
			ServerOpen.TcpIoctl_0.ident 	= tcpINVALID_IDENT
			ServerOpen.TcpIoctl_0.ioctl		= tcpID_LIST_GET
			ServerOpen.TcpIoctl_0.pData		= ADR(IoctlOpenIdents)
			ServerOpen.TcpIoctl_0.datalen 	= SIZEOF(IoctlOpenIdents)
			ServerOpen.TcpIoctl_0 FUB TcpIoctl()

			IF ServerOpen.TcpIoctl_0.status = 0 THEN
				IoctlTotalOpenIdents 	= ServerOpen.TcpIoctl_0.outlen
				IoctlStatus				= ID_Max_Get
			ELSE IF ServerOpen.TcpIoctl_0.status = ERR_FUB_BUSY THEN  (* TcpIoctl not finished -> redo *)
			 	;Busy
			ENDIF
		ELSE IF IoctlStatus = ID_Max_Get THEN
			;Get list of open idents
			ServerOpen.TcpIoctl_0.enable 	= TRUE
			ServerOpen.TcpIoctl_0.ident 	= tcpINVALID_IDENT
			ServerOpen.TcpIoctl_0.ioctl		= tcpID_MAX_GET
			ServerOpen.TcpIoctl_0.pData		= ADR(IoctlMaxIdents)
			ServerOpen.TcpIoctl_0.datalen 	= SIZEOF(IoctlMaxIdents)
			ServerOpen.TcpIoctl_0 FUB TcpIoctl()

			IF ServerOpen.TcpIoctl_0.status = 0 THEN
				IoctlStatus = ID_List_get
			ELSE IF ServerOpen.TcpIoctl_0.status = ERR_FUB_BUSY THEN  (* TcpIoctl not finished -> redo *)
				;Busy
			ENDIF
		ENDIF

	ENDIF

	;Monitor
	IF ServerOpen.Status = sckClosed THEN
		strcpy(ADR(myMonitor.ServerState),"Closed")
	ELSE IF ServerOpen.Status = sckConnecting THEN
		strcpy(ADR(myMonitor.ServerState),"Connecting")
	ELSE IF ServerOpen.Status = sckConnected THEN
		strcpy(ADR(myMonitor.ServerState),"Connected")
	ELSE IF ServerOpen.Status = sckError THEN
		strcpy(ADR(myMonitor.ServerState),"Error")
	ENDIF
	myMonitor.ServerPort 	= ServerOpen.TcpOpen_0.port
	myMonitor.Ident			= ServerOpen.TcpOpen_0.ident

	;Clear Client Connection Counts
	IF ClearConnectCount THEN
		memset(ADR(ClientConnectCount),0,SIZEOF(ClientConnectCount))
		ClearConnectCount = FALSE
	ENDIF

	;Close each connected client connection if open
	LOOP n = 0 TO myMaxConns DO

		IF Server[n].Status = sckError THEN

			Server[n].TcpClose_0.enable 	= TRUE
			Server[n].TcpClose_0.ident 		= Server[n].TcpServer_0.identclnt
			Server[n].TcpClose_0.how 		= 0	; //tcpSHUT_RD OR tcpSHUT_WR;
			Server[n].TcpClose_0 FUB TcpClose()

			IF Server[n].TcpClose_0.status = 0 THEN
				Server[n].Status 				= sckListening
				Server[n].TcpServer_0.identclnt = 0
			ELSE IF Server[n].TcpClose_0.status = tcpERR_INVALID_IDENT THEN
				Server[n].Status 				= sckListening
				Server[n].TcpServer_0.identclnt = 0
			ELSE IF Server[n].TcpClose_0.status = ERR_FUB_BUSY THEN  (* TcpClose not finished -> redo *)
			 	;Busy
			ENDIF

			;Clear the client IP address
			strcpy(ADR(Server[n].client_address),"")
			Server[n].TcpServer_0.portclnt = 0

		ENDIF

		;Listen for a connection
		IF ((Server[n].Status = sckListening) AND (ServerOpen.Status = sckConnected)) THEN

			Server[n].TcpServer_0.enable 	= TRUE							;
			Server[n].TcpServer_0.ident 	= ServerOpen.TcpOpen_0.ident		;  (* Connection Ident from AsTCP.TCP_Open *)
			Server[n].TcpServer_0.backlog 	= 1								;  (* Number of clients waiting simultaneously for a connection*)
			Server[n].TcpServer_0.pIpAddr 	= ADR(Server[n].client_address)	;  (* Where to write the client IP-Address*)
			Server[n].TcpServer_0 FUB TcpServer()											;  (* Call the Function*)

			IF Server[n].TcpServer_0.status = 0 THEN  (* Status = 0 if an client connects to server *)
				Server[n].Status 		= sckSetLinger 	;sckReceive

				;Count then number of connections by any node
				;Check if connected - Client IP address
				Status 		= ethInetAton(ADR(Server[n].client_address),ADR(ClientIP))
				ClientNode 	= 0
				IF (Status = 0) THEN
					;Get the connected node number from the IP address
					Node 		= swapUDINT(ClientIP) ;Mask out the IP address
					ClientNode 	= (Node AND $000000FF)
				ENDIF
				IF ((ClientNode > 0) AND (ClientNode <= 255)) THEN
					ClientConnectCount[ClientNode] = ClientConnectCount[ClientNode] + 1
					IF (ClientConnectCount[ClientNode] > 65000) THEN
						ClearConnectCount = TRUE ;Clear all connections counts whenany connecting client above 65000 times
					ENDIF
				ENDIF

			ELSE IF Server[n].TcpServer_0.status = ERR_FUB_BUSY THEN  (* TcpServer not finished -> redo *)
			  	;Busy
			ENDIF

		ENDIF

		;Set Server Linger Options
		IF Server[n].Status = sckSetLinger THEN

			Server[n].linger_opt.lLinger 	= 0 ;Linger Time = 0
			Server[n].linger_opt.lOnOff		= 1	;Linger Option On

			Server[n].TcpIoctl_0.enable 	= TRUE
			Server[n].TcpIoctl_0.ident 		= Server[n].TcpServer_0.identclnt
			Server[n].TcpIoctl_0.ioctl		= tcpSO_LINGER_SET
			Server[n].TcpIoctl_0.pData		= ADR(Server[n].linger_opt)
			Server[n].TcpIoctl_0.datalen 	= SIZEOF(Server[n].linger_opt)
			Server[n].TcpIoctl_0 FUB TcpIoctl()

			IF Server[n].TcpIoctl_0.status = 0 THEN
				Server[n].Status = sckReceive
			ELSE IF Server[n].TcpIoctl_0.status = ERR_FUB_BUSY THEN  (* TcpIoctl not finished -> redo *)
			 	;Busy
			ENDIF
		ENDIF

		;Receive Data
		IF Server[n].Status = sckReceive THEN

			IF (Server[n].TcpServer_0.identclnt > 0) THEN
				Server[n].TcpRecv_0.enable 		= TRUE
				Server[n].TcpRecv_0.ident 		= Server[n].TcpServer_0.identclnt;  (* Client Ident from AsTCP.TCP_Server *)
				Server[n].TcpRecv_0.pData		= ADR(DisplayData[n].ReceiveData);  (* Where to store the incoming data *)
				Server[n].TcpRecv_0.datamax 	= SIZEOF(DisplayData[n].ReceiveData);  (* Lenght of data buffer *)
				Server[n].TcpRecv_0.flags 		= 0;
				Server[n].TcpRecv_0 FUB TcpRecv()

				IF Server[n].TcpRecv_0.status = 0 THEN  (* Data received *)
					Server[n].Status = sckSend
					Server[n].recv_timeout = 0
				ELSE IF Server[n].TcpRecv_0.status = tcpERR_NO_DATA THEN  (* No data received - wait *)
				   	Server[n].recv_timeout = Server[n].recv_timeout + 1;
				  	IF Server[n].recv_timeout > 50 THEN
		 		    	Server[n].Status 		= sckError
						Server[n].recv_timeout 	= 0
					ENDIF
				ELSE IF Server[n].TcpRecv_0.status = ERR_FUB_BUSY THEN  (* TcpRecv not finished -> redo *)
				 	;Busy
				ELSE IF Server[n].TcpRecv_0.status = tcpERR_NOT_CONNECTED THEN
					Server[n].Status = sckError
				ENDIF
			ELSE
				Server[n].Status = sckError
			ENDIF
		ENDIF

		IF Server[n].Status = sckSend THEN
			IF (Server[n].TcpServer_0.identclnt > 0) THEN
				Server[n].TcpSend_0.enable 		= TRUE
				Server[n].TcpSend_0.ident 		= Server[n].TcpServer_0.identclnt;  (* Client Ident from AsTCP.TCP_Server *)
				Server[n].TcpSend_0.pData 		= ADR(DisplayData[n].SendData);  (* Which data to send *)
				Server[n].TcpSend_0.datalen 	= SIZEOF(DisplayData[n].SendData);  (* Lenght of data to send *)
				Server[n].TcpSend_0.flags 		= 0;
				Server[n].TcpSend_0 FUB TcpSend()

				IF Server[n].TcpSend_0.status = 0 THEN  (* Data sent *)
					Server[n].Status = sckReceive
				ELSE IF Server[n].TcpSend_0.status = ERR_FUB_BUSY THEN  (* TcpSend not finished -> redo *)
				  	;Busy
				ELSE IF (Server[n].TcpSend_0.status = tcpERR_NOT_CONNECTED) THEN
					Server[n].Status = sckError
				ENDIF
			ELSE
				Server[n].Status = sckError
			ENDIF
		ENDIF

		;Copy Client IP to Global Display Data
		DisplayData[n].ClientIP = Server[n].client_address

		;Monitor
		IF Server[n].Status = sckError THEN
			strcpy(ADR(myMonitor.ClientInfo[n].State),"Error")
		ELSE IF Server[n].Status = sckListening THEN
			strcpy(ADR(myMonitor.ClientInfo[n].State),"Listening")
		ELSE IF Server[n].Status = sckReceive THEN
			strcpy(ADR(myMonitor.ClientInfo[n].State),"Receive")
		ELSE IF Server[n].Status = sckSend THEN
			strcpy(ADR(myMonitor.ClientInfo[n].State),"Send")
		ENDIF
		myMonitor.ClientInfo[n].IPAddress 	= Server[n].client_address
		myMonitor.ClientInfo[n].Port 		= Server[n].TcpServer_0.portclnt
		myMonitor.ClientInfo[n].Ident		= Server[n].TcpServer_0.identclnt

	ENDLOOP

END_PROGRAM
```

#### Server.typ - TCP Server Variables
```iecst
(********************************************************************
 * COPYRIGHT -- Bernecker + Rainer
 ********************************************************************
 * Package: LibAsTCP
 * File: LibAsTCP.typ
 * Author: Bernecker + Rainer
 * Created: February 21, 2008
 ********************************************************************
 * Data types of package LibAsTCP
 ********************************************************************)

TYPE
	Monitor_typ : 	STRUCT
		ServerState : STRING[20];
		ServerPort : UINT;
		Ident : UDINT;
		ClientInfo : ARRAY[0..19] OF MonitorClient_typ;
	END_STRUCT;
	MonitorClient_typ : 	STRUCT  (*Monitor selected variables*)
		State : STRING[20];
		Port : UINT;
		IPAddress : STRING[20];
		Ident : UDINT;
	END_STRUCT;
	Server_typ : 	STRUCT  (*TCP Server Variables*)
		Status : USINT; (*TCP Server Connection Status*)
		client_address : STRING[20]; (*Address of the client connection to the Server*)
		TcpServer_0 : TcpServer; (*AsTCP.TcpServer FUB*)
		TcpRecv_0 : TcpRecv; (*AsTCP.TcpRecv FUB*)
		TcpSend_0 : TcpSend; (*AsTCP.TcpSend FUB*)
		TcpClose_0 : TcpClose; (*AsTCP.TcpClose FUB*)
		TcpIoctl_0 : TcpIoctl; (*AsTCP.TcpIoctl*)
		linger_opt : tcpLINGER_typ;
		recv_timeout : UDINT; (*receive timeout*)
	END_STRUCT;
	ServerOpen_typ : 	STRUCT
		Status : UINT;
		linger_opt : tcpLINGER_typ;
		TcpIoctl_0 : TcpIoctl; (*AsTCP.TcpIoctl*)
		TcpOpen_0 : TcpOpen; (*AsTCP.TcpOpen FUB*)
		TcpClose_0 : TcpClose; (*AsTCP.TcpClose FUB*)
	END_STRUCT;
END_TYPE
```

#### Server.var - Data for Server Task
```iecst
(********************************************************************
 * COPYRIGHT -- Bernecker + Rainer
 ********************************************************************
 * Package: LibAsTCP
 * File: LibAsTCP.var
 * Author: Bernecker + Rainer
 * Created: February 21, 2008
 ********************************************************************
 * Variables of package LibAsTCP
 ********************************************************************)
VAR
	data_buffer : ARRAY[0..100] OF UDINT;
END_VAR
VAR CONSTANT
	sckClosed : USINT := 0;
	sckConnecting : USINT := 1;
	sckConnected : USINT := 2;
	sckError : USINT := 3;
	sckListening : USINT := 4;
	sckReceive : USINT := 5;
	sckSend : USINT := 6;
	sckSetLinger : USINT := 7;
END_VAR
VAR
	Server : ARRAY[0..19] OF Server_typ; (*Data for Server Task*)
	ServerOpen : ServerOpen_typ;
END_VAR
VAR RETAIN
	IdentRetain : UDINT;
END_VAR
VAR
	n : UINT;
	ServerSize : UDINT;
	mySize : UINT;
	myMaxConns : UINT;
	myMonitor : Monitor_typ;
	TON_10ms_0 : TON_10ms;
	Index : UINT;
	IoctlOpenIdents : ARRAY[0..49] OF UDINT;
	IoctlTotalOpenIdents : UDINT;
	IoctlMaxIdents : UDINT;
	IoctlStatus : UINT;
	ID_List_get : UINT := 0;
	ID_Max_Get : UINT := 1;
	ClientNode : UDINT;
	Status : UINT;
	ClientIP : UDINT;
	Node : UDINT;
	ClientConnectCount : ARRAY[0..255] OF UINT;
	ClearConnectCount : BOOL;
END_VAR
```

### Program Logical/Displays/zzClientText (IEC, version 1.01.1) - AsTCP Diplay Client

#### Client.ab - Implementation code
```automation-basic
(********************************************************************
 * COPYRIGHT --
 ********************************************************************
 * PROGRAM: Client
 * File: Client.ab
 * Author: Dave
 * Created: December 06, 2010
 ********************************************************************
 * Implementation OF PROGRAM Client
 ********************************************************************)

;Version 1.00 12/12/2010 D.J. First Issue
;Version 1.01.0 12/07/2016 - TR Fix issue not clearing bag data
;Version 1.01.1 16/08/2017	- TR- Fix issue with random data loss.

PROGRAM _INIT

END_PROGRAM

PROGRAM _CYCLIC
	mySql = 75

	SQL.Login	= ClientReceive[0].SQL
	IF NOT WaitReply THEN

		myQuad = myQuad + 2
		IF (myQuad > 2) THEN
			myQuad = 0
		ENDIF

		IF (ClientText[myQuad].Cat <> ClientReceive[myQuad].DisplayBag.Cat) THEN
			strcpy(ADR(ClientText[myQuad].CatName),"")
			strcpy(ADR(ClientText[myQuad].CatLong),"")
			strcpy(ADR(ClientText[myQuad].ImagePath),"")
			ClientText[myQuad].Cat = 0;
			ClientText[myQuad].Prg = 0
			WaitReply = (ClientReceive[myQuad].DisplayBag.Cat > 0)
		ENDIF

		IF (ClientText[myQuad].Cus <> ClientReceive[myQuad].DisplayBag.Cus) THEN
			strcpy(ADR(ClientText[myQuad].CusName),"")
			strcpy(ADR(ClientText[myQuad].CusLong),"")
			ClientText[myQuad].Cus = 0
			WaitReply = ((ClientReceive[myQuad].DisplayBag.Cus > 0) OR WaitReply)
		ENDIF

		IF (ClientText[myQuad + 1].Cat <> ClientReceive[myQuad + 1].DisplayBag.Cat) THEN
			strcpy(ADR(ClientText[myQuad + 1].CatName),"")
			strcpy(ADR(ClientText[myQuad + 1].CatLong),"")
			strcpy(ADR(ClientText[myQuad + 1].ImagePath),"")
			ClientText[myQuad + 1].Cat = 0;
			ClientText[myQuad + 1].Prg = 0
			WaitReply = ((ClientReceive[myQuad + 1].DisplayBag.Cat > 0) OR WaitReply)
		ENDIF

		IF (ClientText[myQuad + 1].Cus <> ClientReceive[myQuad + 1].DisplayBag.Cus) THEN
			strcpy(ADR(ClientText[myQuad + 1].CusName),"")
			strcpy(ADR(ClientText[myQuad + 1].CusLong),"")
			ClientText[myQuad + 1].Cus = 0
			WaitReply =  ((ClientReceive[myQuad + 1].DisplayBag.Cus > 0) OR WaitReply)
		ENDIF
		;Set TrackView Registers
		IF WaitReply THEN
			itoa(ClientReceive[myQuad].DisplayBag.Cat,ADR(myCatString))
			itoa(ClientReceive[myQuad].DisplayBag.Cus,ADR(myCusString))
			itoa(ClientReceive[myQuad + 1].DisplayBag.Cat,ADR(myCatString1))
			itoa(ClientReceive[myQuad + 1].DisplayBag.Cus,ADR(myCusString1))

			SqlRequest[mySql].Request = TRUE
		ENDIF

	ENDIF

	;Set request to TrackView until reply
	IF (WaitReply AND SqlRequest[mySql].Complete) THEN

		ClientText[myQuad].Prg = USINT(atoi(ADR(SqlRequest[mySql].OutputData[1])))
		strcpy(ADR(ClientText[myQuad].PrgLong),ADR(SqlRequest[mySql].OutputData[2]))
		strcpy(ADR(ClientText[myQuad].PrgName),ADR(SqlRequest[mySql].OutputData[3]))

		;		strcpy(ADR(ClientText[myQuad].CatName),"")
		;		strcpy(ADR(ClientText[myQuad].CatLong),"")
		;		strcpy(ADR(ClientText[myQuad].ImagePath),"")

		ClientText[myQuad].Cat = atoi(ADR(SqlRequest[mySql].Parameters[0].Param_String))
		strcpy(ADR(ClientText[myQuad].CatLong),ADR(SqlRequest[mySql].OutputData[4]))
		strcpy(ADR(ClientText[myQuad].CatName),ADR(SqlRequest[mySql].OutputData[5]))

		;		strcpy(ADR(ClientText[myQuad].Cus),"")
		;		strcpy(ADR(ClientText[myQuad].CusLong),"")

		ClientText[myQuad].Cus = atoi(ADR(SqlRequest[mySql].Parameters[1].Param_String))
		strcpy(ADR(ClientText[myQuad].CusLong),ADR(SqlRequest[mySql].OutputData[6]))
		strcpy(ADR(ClientText[myQuad].CusName),ADR(SqlRequest[mySql].OutputData[7]))

		strcpy(ADR(ClientText[myQuad].ImagePath),ADR(SqlRequest[mySql].OutputData[8]))

		ClientText[myQuad + 1].Prg = USINT(atoi(ADR(SqlRequest[mySql].OutputData[9])))
		strcpy(ADR(ClientText[myQuad + 1].PrgLong),ADR(SqlRequest[mySql].OutputData[10]))
		strcpy(ADR(ClientText[myQuad + 1].PrgName),ADR(SqlRequest[mySql].OutputData[11]))

		;		strcpy(ADR(ClientText[myQuad + 1].CatName),"")
		;		strcpy(ADR(ClientText[myQuad + 1].CatLong),"")
		;		strcpy(ADR(ClientText[myQuad + 1].ImagePath),"")

		ClientText[myQuad + 1].Cat = atoi(ADR(SqlRequest[mySql].Parameters[2].Param_String))
		strcpy(ADR(ClientText[myQuad + 1].CatLong),ADR(SqlRequest[mySql].OutputData[12]))
		strcpy(ADR(ClientText[myQuad + 1].CatName),ADR(SqlRequest[mySql].OutputData[13]))

		;		strcpy(ADR(ClientText[myQuad].Cus),"")
		;		strcpy(ADR(ClientText[myQuad].CusLong),"")

		ClientText[myQuad + 1].Cus = atoi(ADR(SqlRequest[mySql].Parameters[3].Param_String))
		strcpy(ADR(ClientText[myQuad + 1].CusLong),ADR(SqlRequest[mySql].OutputData[14]))
		strcpy(ADR(ClientText[myQuad + 1].CusName),ADR(SqlRequest[mySql].OutputData[15]))

		strcpy(ADR(ClientText[myQuad + 1].ImagePath),ADR(SqlRequest[mySql].OutputData[16]))

		WaitReply 	= FALSE

	ENDIF

	IF SqlRequest[mySql].Request AND NOT SqlWriteActive THEN ; Write Count to SQL
		SqlWriteActive = TRUE
		SqlRequest[mySql].SQLType = cSQLType_ReadWrite
		SqlRequest[mySql].SQL_usp = cSQLReq_zzGetMultiNames
		SqlRequest[mySql].NoOfParams = 4

		SqlRequest[mySql].Parameters[0].Type = cSQLParam_Input ;
		strcpy(ADR(SqlRequest[mySql].Parameters[0].Param_String),ADR(myCatString))
		SqlRequest[mySql].Parameters[1].Type = cSQLParam_Input ;
		strcpy(ADR(SqlRequest[mySql].Parameters[1].Param_String),ADR(myCusString))
		SqlRequest[mySql].Parameters[2].Type = cSQLParam_Input ;
		strcpy(ADR(SqlRequest[mySql].Parameters[2].Param_String),ADR(myCatString1))
		SqlRequest[mySql].Parameters[3].Type = cSQLParam_Input ;
		strcpy(ADR(SqlRequest[mySql].Parameters[3].Param_String),ADR(myCusString1))
	ENDIF

	IF SqlRequest[mySql].Complete THEN ; ClearRequest
		;Copy Out Reply Done in step.!
		SqlRequest[mySql] = cEmptySQlReq
		SqlWriteActive = FALSE
	ELSE IF SqlRequest[mySql].Fail THEN
		WaitReply = FALSE ; Move to next and try and again
		SqlWriteActive = FALSE ; Reload Parameters
		SqlRequest[mySql].Fail = FALSE
	ENDIF
END_PROGRAM
```

#### Client.var - Local variables
```iecst
VAR
	myQuad : UINT;
	WaitReply : BOOL;
	myCatString : STRING[11];
	myCusString : STRING[11];
	mySql : USINT;
	SqlWriteActive : BOOL;
	myCatString1 : STRING[11];
	myCusString1 : STRING[11];
END_VAR
```

### Program Logical/Displays/ClientPanel (IEC, version 2.00.0) - Client Panel Control
